LIN {X 0,Y 483.427,Z 781.933,A -85,B 0,C 180,E1 -6916.12,E2 -6916.12} C_VEL
LIN {X 0,Y 482.975,Z 793.62,A -85,B 0,C 180,E1 -6916.772,E2 -6916.772} C_VEL
LIN {X 0,Y 482.538,Z 805.095,A -85,B 0,C 180,E1 -6917.594,E2 -6917.594} C_VEL
LIN {X 0,Y 482.15,Z 815.757,A -85,B 0,C 180,E1 -6918.544,E2 -6918.544} C_VEL
LIN {X 0,Y 481.803,Z 824.454,A -85,B 0,C 180,E1 -6919.494,E2 -6919.494} C_VEL
LIN {X 0,Y 481.522,Z 832.495,A -85,B 0,C 180,E1 -6920.549,E2 -6920.549} C_VEL
LIN {X 0,Y 481.338,Z 839.236,A -85,B 0,C 180,E1 -6921.604,E2 -6921.604} C_VEL
LIN {X 0,Y 481.117,Z 845.911,A -85,B 0,C 180,E1 -6922.867,E2 -6922.867} C_VEL
LIN {X 0,Y 481.068,Z 851.207,A -85,B 0,C 180,E1 -6924.13,E2 -6924.13} C_VEL
LIN {X 0,Y 480.941,Z 855.277,A -85,B 0,C 180,E1 -6925.39,E2 -6925.39} C_VEL
LIN {X 0,Y 480.957,Z 858.306,A -85,B 0,C 180,E1 -6926.649,E2 -6926.649} C_VEL
LIN {X 0,Y 480.902,Z 859.812,A -85,B 0,C 180,E1 -6927.487,E2 -6927.487} C_VEL
LIN {X 0,Y 480.86,Z 861.418,A -85,B 0,C 180,E1 -6929.162,E2 -6929.162} C_VEL
LIN {X 0,Y 480.844,Z 861.684,A -85,B 0,C 180,E1 -6930,E2 -6930} C_VEL
LIN {X 0,Y 480.855,Z 861.455,A -85,B 0,C 180,E1 -6930.837,E2 -6930.837} C_VEL
LIN {X 0,Y 480.902,Z 859.817,A -85,B 0,C 180,E1 -6932.512,E2 -6932.512} C_VEL
LIN {X 0,Y 480.955,Z 858.409,A -85,B 0,C 180,E1 -6933.35,E2 -6933.35} C_VEL
LIN {X 0,Y 480.94,Z 855.356,A -85,B 0,C 180,E1 -6934.609,E2 -6934.609} C_VEL
LIN {X 0,Y 481.067,Z 851.27,A -85,B 0,C 180,E1 -6935.869,E2 -6935.869} C_VEL
LIN {X 0,Y 481.15,Z 845.081,A -85,B 0,C 180,E1 -6937.342,E2 -6937.342} C_VEL
LIN {X 0,Y 481.372,Z 838.203,A -85,B 0,C 180,E1 -6938.606,E2 -6938.606} C_VEL
LIN {X 0,Y 481.64,Z 829.782,A -85,B 0,C 180,E1 -6939.872,E2 -6939.872} C_VEL
LIN {X 0,Y 481.945,Z 821.073,A -85,B 0,C 180,E1 -6940.927,E2 -6940.927} C_VEL
LIN {X 0,Y 482.433,Z 810.454,A -85,B 0,C 180,E1 -6941.981,E2 -6941.981} C_VEL
LIN {X 0,Y 482.803,Z 798.946,A -85,B 0,C 180,E1 -6942.9,E2 -6942.9} C_VEL
LIN {X 0,Y 483.277,Z 786.489,A -85,B 0,C 180,E1 -6943.669,E2 -6943.669} C_VEL
LIN {X 0,Y 483.656,Z 774.047,A -85,B 0,C 180,E1 -6944.247,E2 -6944.247} C_VEL
LIN {X 0,Y 483.668,Z 767.501,A -85,B 0,C 180,E1 -6944.489,E2 -6944.489} C_VEL
LIN {X 0,Y 482.005,Z 754.779,A -85,B 0,C 180,E1 -6944.877,E2 -6944.877} C_VEL
LIN {X 0,Y 481.559,Z 749.951,A -85,B 0,C 180,E1 -6944.986,E2 -6944.986} C_VEL
LIN {X 0,Y 481.886,Z 734.845,A -85,B 0,C 180,E1 -6948.206,E2 -6948.206} C_VEL
LIN {X 0,Y 482.217,Z 720.246,A -85,B 0,C 180,E1 -6951.367,E2 -6951.367} C_VEL
LIN {X 0,Y 482.622,Z 704.896,A -85,B 0,C 180,E1 -6954.749,E2 -6954.749} C_VEL
LIN {X 0,Y 483.035,Z 691.607,A -85,B 0,C 180,E1 -6957.748,E2 -6957.748} C_VEL
LIN {X 0,Y 483.624,Z 676.701,A -85,B 0,C 180,E1 -6961.205,E2 -6961.205} C_VEL
LIN {X 0,Y 484.172,Z 663.094,A -85,B 0,C 180,E1 -6964.478,E2 -6964.478} C_VEL
LIN {X 0,Y 484.454,Z 654.94,A -85,B 0,C 180,E1 -6966.497,E2 -6966.497} C_VEL
LIN {X 0,Y 482.901,Z 646.667,A -85,B 0,C 180,E1 -6968.741,E2 -6968.741} C_VEL
LIN {X 0,Y 481.668,Z 640.49,A -85,B 0,C 180,E1 -6970.52,E2 -6970.52} C_VEL
LIN {X 0,Y 481.637,Z 640.491,A -85,B 0,C 180,E1 -6973.299,E2 -6973.299} C_VEL
LIN {X 0,Y 481.682,Z 640.488,A -85,B 0,C 180,E1 -6976.705,E2 -6976.705} C_VEL
LIN {X 0,Y 481.69,Z 640.485,A -85,B 0,C 180,E1 -6980.061,E2 -6980.061} C_VEL
LIN {X 0,Y 481.634,Z 640.491,A -85,B 0,C 180,E1 -6982.203,E2 -6982.203} C_VEL
LIN {X 0,Y 481.688,Z 640.479,A -85,B 0,C 180,E1 -6985.318,E2 -6985.318} C_VEL
LIN {X 0,Y 481.644,Z 640.487,A -85,B 0,C 180,E1 -6988.311,E2 -6988.311} C_VEL
LIN {X 0,Y 481.703,Z 640.479,A -85,B 0,C 180,E1 -6991.219,E2 -6991.219} C_VEL
LIN {X 0,Y 481.702,Z 640.479,A -85,B 0,C 180,E1 -6994.043,E2 -6994.043} C_VEL
LIN {X 0,Y 481.67,Z 640.483,A -85,B 0,C 180,E1 -6996.811,E2 -6996.811} C_VEL
LIN {X 0,Y 481.692,Z 640.483,A -85,B 0,C 180,E1 -6999.502,E2 -6999.502} C_VEL
LIN {X 0,Y 481.702,Z 640.478,A -85,B 0,C 180,E1 -7002.158,E2 -7002.158} C_VEL
LIN {X 0,Y 481.737,Z 640.479,A -85,B 0,C 180,E1 -7004.775,E2 -7004.775} C_VEL
LIN {X 0,Y 481.791,Z 640.47,A -85,B 0,C 180,E1 -7008.216,E2 -7008.216} C_VEL
LIN {X 0,Y 481.759,Z 640.473,A -85,B 0,C 180,E1 -7011.611,E2 -7011.611} C_VEL
LIN {X 0,Y 481.811,Z 640.47,A -85,B 0,C 180,E1 -7014.139,E2 -7014.139} C_VEL
LIN {X 0,Y 481.923,Z 640.453,A -85,B 0,C 180,E1 -7017.492,E2 -7017.492} C_VEL
LIN {X 0,Y 481.9,Z 640.459,A -85,B 0,C 180,E1 -7020.836,E2 -7020.836} C_VEL
LIN {X 0,Y 481.924,Z 640.458,A -85,B 0,C 180,E1 -7022.507,E2 -7022.507} C_VEL
LIN {X 0,Y 481.743,Z 640.595,A -85,B 0,C 180,E1 -7023.555,E2 -7023.555} C_VEL
LIN {X 0,Y 482.624,Z 646.304,A -85,B 0,C 180,E1 -7025.012,E2 -7025.012} C_VEL
LIN {X 0,Y 482.79,Z 656.329,A -85,B 0,C 180,E1 -7027.528,E2 -7027.528} C_VEL
LIN {X 0,Y 482.659,Z 667.926,A -85,B 0,C 180,E1 -7030.487,E2 -7030.487} C_VEL
LIN {X 0,Y 482.588,Z 677.613,A -85,B 0,C 180,E1 -7033.003,E2 -7033.003} C_VEL
LIN {X 0,Y 482.37,Z 689.295,A -85,B 0,C 180,E1 -7036.071,E2 -7036.071} C_VEL
LIN {X 0,Y 482.136,Z 700.788,A -85,B 0,C 180,E1 -7039.146,E2 -7039.146} C_VEL
LIN {X 0,Y 481.9,Z 712.481,A -85,B 0,C 180,E1 -7042.283,E2 -7042.283} C_VEL
LIN {X 0,Y 481.666,Z 724.354,A -85,B 0,C 180,E1 -7045.504,E2 -7045.504} C_VEL
LIN {X 0,Y 481.595,Z 726.474,A -85,B 0,C 180,E1 -7046.079,E2 -7046.079} C_VEL
LIN {X 0,Y 484.069,Z 741.262,A -85,B 0,C 180,E1 -7046.545,E2 -7046.545} C_VEL
LIN {X 0,Y 483.708,Z 754.433,A -85,B 0,C 180,E1 -7047.052,E2 -7047.052} C_VEL
LIN {X 0,Y 483.248,Z 767.048,A -85,B 0,C 180,E1 -7047.735,E2 -7047.735} C_VEL
LIN {X 0,Y 482.824,Z 779.115,A -85,B 0,C 180,E1 -7048.589,E2 -7048.589} C_VEL
LIN {X 0,Y 482.382,Z 789.501,A -85,B 0,C 180,E1 -7049.524,E2 -7049.524} C_VEL
LIN {X 0,Y 481.935,Z 799.526,A -85,B 0,C 180,E1 -7050.641,E2 -7050.641} C_VEL
LIN {X 0,Y 481.601,Z 807.216,A -85,B 0,C 180,E1 -7051.692,E2 -7051.692} C_VEL
LIN {X 0,Y 481.345,Z 814.641,A -85,B 0,C 180,E1 -7052.932,E2 -7052.932} C_VEL
LIN {X 0,Y 481.11,Z 820.823,A -85,B 0,C 180,E1 -7054.222,E2 -7054.222} C_VEL
LIN {X 0,Y 480.916,Z 826.562,A -85,B 0,C 180,E1 -7055.771,E2 -7055.771} C_VEL
LIN {X 0,Y 480.832,Z 829.462,A -85,B 0,C 180,E1 -7056.818,E2 -7056.818} C_VEL
LIN {X 0,Y 480.783,Z 831.725,A -85,B 0,C 180,E1 -7057.875,E2 -7057.875} C_VEL
LIN {X 0,Y 480.702,Z 833.614,A -85,B 0,C 180,E1 -7059.208,E2 -7059.208} C_VEL
LIN {X 0,Y 480.658,Z 834.484,A -85,B 0,C 180,E1 -7060.508,E2 -7060.508} C_VEL
LIN {X 0,Y 480.685,Z 834.413,A -85,B 0,C 180,E1 -7061.785,E2 -7061.785} C_VEL
LIN {X 0,Y 480.698,Z 832.973,A -85,B 0,C 180,E1 -7063.406,E2 -7063.406} C_VEL
LIN {X 0,Y 480.847,Z 830.113,A -85,B 0,C 180,E1 -7064.998,E2 -7064.998} C_VEL
LIN {X 0,Y 480.928,Z 826.941,A -85,B 0,C 180,E1 -7066.185,E2 -7066.185} C_VEL
LIN {X 0,Y 481.052,Z 822.862,A -85,B 0,C 180,E1 -7067.36,E2 -7067.36} C_VEL
LIN {X 0,Y 481.177,Z 817.743,A -85,B 0,C 180,E1 -7068.539,E2 -7068.539} C_VEL
LIN {X 0,Y 481.468,Z 810.441,A -85,B 0,C 180,E1 -7069.883,E2 -7069.883} C_VEL
LIN {X 0,Y 481.805,Z 801.756,A -85,B 0,C 180,E1 -7071.155,E2 -7071.155} C_VEL
LIN {X 0,Y 482.202,Z 792.467,A -85,B 0,C 180,E1 -7072.256,E2 -7072.256} C_VEL
LIN {X 0,Y 482.643,Z 782.457,A -85,B 0,C 180,E1 -7073.214,E2 -7073.214} C_VEL
LIN {X 0,Y 483.059,Z 771.967,A -85,B 0,C 180,E1 -7074.027,E2 -7074.027} C_VEL
LIN {X 0,Y 483.552,Z 759.705,A -85,B 0,C 180,E1 -7074.774,E2 -7074.774} C_VEL
LIN {X 0,Y 483.802,Z 750.922,A -85,B 0,C 180,E1 -7075.188,E2 -7075.188} C_VEL
LIN {X 0,Y 483.217,Z 747.306,A -85,B 0,C 180,E1 -7075.36,E2 -7075.36} C_VEL
LIN {X 0,Y 481.631,Z 743.95,A -85,B 0,C 180,E1 -7075.54,E2 -7075.54} C_VEL
LIN {X 0,Y 476.928,Z 736.321,A -85,B 0,C 180,E1 -7075.926,E2 -7075.926} C_VEL
LIN {X 0,Y 475.668,Z 732.622,A -85,B 0,C 180,E1 -7076.054,E2 -7076.054} C_VEL
LIN {X 0,Y 474.549,Z 726.5,A -85,B 0,C 180,E1 -7076.238,E2 -7076.238} C_VEL
LIN {X 0,Y 474.82,Z 714.749,A -85,B 0,C 180,E1 -7079.469,E2 -7079.469} C_VEL
LIN {X 0,Y 475.098,Z 704.87,A -85,B 0,C 180,E1 -7082.202,E2 -7082.202} C_VEL
LIN {X 0,Y 475.378,Z 694.436,A -85,B 0,C 180,E1 -7085.081,E2 -7085.081} C_VEL
LIN {X 0,Y 475.689,Z 682.671,A -85,B 0,C 180,E1 -7088.325,E2 -7088.325} C_VEL
LIN {X 0,Y 475.933,Z 671.182,A -85,B 0,C 180,E1 -7091.49,E2 -7091.49} C_VEL
LIN {X 0,Y 476.149,Z 659.898,A -85,B 0,C 180,E1 -7094.593,E2 -7094.593} C_VEL
LIN {X 0,Y 476.103,Z 650.411,A -85,B 0,C 180,E1 -7097.208,E2 -7097.208} C_VEL
LIN {X 0,Y 475.298,Z 644.411,A -85,B 0,C 180,E1 -7098.918,E2 -7098.918} C_VEL
LIN {X 0,Y 474.693,Z 641.359,A -85,B 0,C 180,E1 -7099.821,E2 -7099.821} C_VEL
LIN {X 0,Y 474.786,Z 641.347,A -85,B 0,C 180,E1 -7102.642,E2 -7102.642} C_VEL
LIN {X 0,Y 474.755,Z 641.351,A -85,B 0,C 180,E1 -7104.905,E2 -7104.905} C_VEL
LIN {X 0,Y 474.896,Z 641.333,A -85,B 0,C 180,E1 -7107.456,E2 -7107.456} C_VEL
LIN {X 0,Y 474.914,Z 641.329,A -85,B 0,C 180,E1 -7110,E2 -7110} C_VEL
LIN {X 0,Y 474.896,Z 641.331,A -85,B 0,C 180,E1 -7112.545,E2 -7112.545} C_VEL
LIN {X 0,Y 474.772,Z 641.348,A -85,B 0,C 180,E1 -7115.948,E2 -7115.948} C_VEL
LIN {X 0,Y 474.73,Z 641.353,A -85,B 0,C 180,E1 -7118.514,E2 -7118.514} C_VEL
LIN {X 0,Y 474.741,Z 641.349,A -85,B 0,C 180,E1 -7121.962,E2 -7121.962} C_VEL
LIN {X 0,Y 474.683,Z 641.358,A -85,B 0,C 180,E1 -7125.768,E2 -7125.768} C_VEL
LIN {X 0,Y 474.667,Z 641.361,A -85,B 0,C 180,E1 -7129.01,E2 -7129.01} C_VEL
LIN {X 0,Y 474.589,Z 641.371,A -85,B 0,C 180,E1 -7131.729,E2 -7131.729} C_VEL
LIN {X 0,Y 474.649,Z 641.364,A -85,B 0,C 180,E1 -7133.652,E2 -7133.652} C_VEL
LIN {X 0,Y 477.203,Z 650.814,A -85,B 0,C 180,E1 -7134.238,E2 -7134.238} C_VEL
LIN {X 0,Y 476.972,Z 661.909,A -85,B 0,C 180,E1 -7134.947,E2 -7134.947} C_VEL
LIN {X 0,Y 476.498,Z 673.39,A -85,B 0,C 180,E1 -7135.881,E2 -7135.881} C_VEL
LIN {X 0,Y 476.09,Z 683.215,A -85,B 0,C 180,E1 -7136.878,E2 -7136.878} C_VEL
LIN {X 0,Y 475.726,Z 692.476,A -85,B 0,C 180,E1 -7138.038,E2 -7138.038} C_VEL
LIN {X 0,Y 475.342,Z 700.4,A -85,B 0,C 180,E1 -7139.27,E2 -7139.27} C_VEL
LIN {X 0,Y 475.043,Z 706.99,A -85,B 0,C 180,E1 -7140.538,E2 -7140.538} C_VEL
LIN {X 0,Y 474.802,Z 711.876,A -85,B 0,C 180,E1 -7141.7,E2 -7141.7} C_VEL
LIN {X 0,Y 474.595,Z 716.839,A -85,B 0,C 180,E1 -7143.224,E2 -7143.224} C_VEL
LIN {X 0,Y 474.467,Z 719.337,A -85,B 0,C 180,E1 -7144.255,E2 -7144.255} C_VEL
LIN {X 0,Y 474.365,Z 721.447,A -85,B 0,C 180,E1 -7145.427,E2 -7145.427} C_VEL
LIN {X 0,Y 474.285,Z 722.963,A -85,B 0,C 180,E1 -7146.853,E2 -7146.853} C_VEL
LIN {X 0,Y 474.312,Z 723.349,A -85,B 0,C 180,E1 -7148.486,E2 -7148.486} C_VEL
LIN {X 0,Y 474.353,Z 722.79,A -85,B 0,C 180,E1 -7149.607,E2 -7149.607} C_VEL
LIN {X 0,Y 474.425,Z 721.256,A -85,B 0,C 180,E1 -7150.931,E2 -7150.931} C_VEL
LIN {X 0,Y 474.576,Z 718.785,A -85,B 0,C 180,E1 -7152.23,E2 -7152.23} C_VEL
LIN {X 0,Y 474.751,Z 715.391,A -85,B 0,C 180,E1 -7153.5,E2 -7153.5} C_VEL
LIN {X 0,Y 474.957,Z 710.197,A -85,B 0,C 180,E1 -7154.952,E2 -7154.952} C_VEL
LIN {X 0,Y 475.317,Z 703.304,A -85,B 0,C 180,E1 -7156.428,E2 -7156.428} C_VEL
LIN {X 0,Y 475.677,Z 696.215,A -85,B 0,C 180,E1 -7157.624,E2 -7157.624} C_VEL
LIN {X 0,Y 476.057,Z 687.294,A -85,B 0,C 180,E1 -7158.843,E2 -7158.843} C_VEL
LIN {X 0,Y 476.534,Z 678.215,A -85,B 0,C 180,E1 -7159.848,E2 -7159.848} C_VEL
LIN {X 0,Y 476.893,Z 668.033,A -85,B 0,C 180,E1 -7160.769,E2 -7160.769} C_VEL
LIN {X 0,Y 477.24,Z 656.015,A -85,B 0,C 180,E1 -7161.62,E2 -7161.62} C_VEL
LIN {X 0,Y 477.318,Z 650.683,A -85,B 0,C 180,E1 -7161.934,E2 -7161.934} C_VEL
LIN {X 0,Y 474.626,Z 641.364,A -85,B 0,C 180,E1 -7162.519,E2 -7162.519} C_VEL
LIN {X 0,Y 474.638,Z 641.362,A -85,B 0,C 180,E1 -7166.016,E2 -7166.016} C_VEL
LIN {X 0,Y 474.605,Z 641.367,A -85,B 0,C 180,E1 -7169.19,E2 -7169.19} C_VEL
LIN {X 0,Y 474.647,Z 641.365,A -85,B 0,C 180,E1 -7171.718,E2 -7171.718} C_VEL
LIN {X 0,Y 474.652,Z 641.356,A -85,B 0,C 180,E1 -7174.583,E2 -7174.583} C_VEL
LIN {X 0,Y 474.601,Z 641.362,A -85,B 0,C 180,E1 -7177.355,E2 -7177.355} C_VEL
LIN {X 0,Y 474.656,Z 641.361,A -85,B 0,C 180,E1 -7180.09,E2 -7180.09} C_VEL
LIN {X 0,Y 474.651,Z 641.356,A -85,B 0,C 180,E1 -7182.775,E2 -7182.775} C_VEL
LIN {X 0,Y 474.649,Z 641.36,A -85,B 0,C 180,E1 -7185.421,E2 -7185.421} C_VEL
LIN {X 0,Y 474.705,Z 641.354,A -85,B 0,C 180,E1 -7188.038,E2 -7188.038} C_VEL
LIN {X 0,Y 474.729,Z 641.349,A -85,B 0,C 180,E1 -7191.487,E2 -7191.487} C_VEL
LIN {X 0,Y 474.78,Z 641.347,A -85,B 0,C 180,E1 -7194.053,E2 -7194.053} C_VEL
LIN {X 0,Y 474.896,Z 641.323,A -85,B 0,C 180,E1 -7197.456,E2 -7197.456} C_VEL
LIN {X 0,Y 474.913,Z 641.328,A -85,B 0,C 180,E1 -7200,E2 -7200} C_VEL
LIN {X 0,Y 474.896,Z 641.328,A -85,B 0,C 180,E1 -7202.545,E2 -7202.545} C_VEL
LIN {X 0,Y 474.78,Z 641.341,A -85,B 0,C 180,E1 -7205.948,E2 -7205.948} C_VEL
LIN {X 0,Y 474.73,Z 641.346,A -85,B 0,C 180,E1 -7208.514,E2 -7208.514} C_VEL
LIN {X 0,Y 474.706,Z 641.354,A -85,B 0,C 180,E1 -7211.963,E2 -7211.963} C_VEL
LIN {X 0,Y 474.701,Z 641.35,A -85,B 0,C 180,E1 -7215.456,E2 -7215.456} C_VEL
LIN {X 0,Y 474.666,Z 641.354,A -85,B 0,C 180,E1 -7219.01,E2 -7219.01} C_VEL
LIN {X 0,Y 474.59,Z 641.365,A -85,B 0,C 180,E1 -7221.729,E2 -7221.729} C_VEL
LIN {X 0,Y 474.659,Z 641.362,A -85,B 0,C 180,E1 -7224.493,E2 -7224.493} C_VEL
LIN {X 0,Y 474.683,Z 641.353,A -85,B 0,C 180,E1 -7227.334,E2 -7227.334} C_VEL
LIN {X 0,Y 474.607,Z 641.367,A -85,B 0,C 180,E1 -7230.23,E2 -7230.23} C_VEL
LIN {X 0,Y 474.645,Z 641.36,A -85,B 0,C 180,E1 -7233.22,E2 -7233.22} C_VEL
LIN {X 0,Y 474.591,Z 641.371,A -85,B 0,C 180,E1 -7236.324,E2 -7236.324} C_VEL
LIN {X 0,Y 474.63,Z 641.361,A -85,B 0,C 180,E1 -7239.648,E2 -7239.648} C_VEL
LIN {X 0,Y 474.618,Z 641.363,A -85,B 0,C 180,E1 -7242.934,E2 -7242.934} C_VEL
LIN {X 0,Y 474.612,Z 641.365,A -85,B 0,C 180,E1 -7245.895,E2 -7245.895} C_VEL
LIN {X 0,Y 474.63,Z 641.372,A -85,B 0,C 180,E1 -7249.041,E2 -7249.041} C_VEL
LIN {X 0,Y 474.648,Z 641.378,A -85,B 0,C 180,E1 -7249.799,E2 -7249.799} C_VEL
LIN {X 0,Y 476.716,Z 652.009,A -85,B 0,C 180,E1 -7252.811,E2 -7252.811} C_VEL
LIN {X 0,Y 477.086,Z 656.071,A -85,B 0,C 180,E1 -7253.896,E2 -7253.896} C_VEL
LIN {X 0,Y 476.52,Z 669.453,A -85,B 0,C 180,E1 -7257.211,E2 -7257.211} C_VEL
LIN {X 0,Y 476.074,Z 682.373,A -85,B 0,C 180,E1 -7260.276,E2 -7260.276} C_VEL
LIN {X 0,Y 475.643,Z 697.254,A -85,B 0,C 180,E1 -7263.687,E2 -7263.687} C_VEL
LIN {X 0,Y 475.306,Z 709.747,A -85,B 0,C 180,E1 -7266.47,E2 -7266.47} C_VEL
LIN {X 0,Y 474.934,Z 725.361,A -85,B 0,C 180,E1 -7269.876,E2 -7269.876} C_VEL
LIN {X 0,Y 474.656,Z 738.834,A -85,B 0,C 180,E1 -7272.774,E2 -7272.774} C_VEL
LIN {X 0,Y 474.456,Z 748.246,A -85,B 0,C 180,E1 -7274.783,E2 -7274.783} C_VEL
LIN {X 0,Y 475.885,Z 762.604,A -85,B 0,C 180,E1 -7275.172,E2 -7275.172} C_VEL
LIN {X 0,Y 476.883,Z 769.641,A -85,B 0,C 180,E1 -7275.436,E2 -7275.436} C_VEL
LIN {X 0,Y 476.45,Z 781.864,A -85,B 0,C 180,E1 -7275.968,E2 -7275.968} C_VEL
LIN {X 0,Y 475.937,Z 794.279,A -85,B 0,C 180,E1 -7276.692,E2 -7276.692} C_VEL
LIN {X 0,Y 475.441,Z 808.391,A -85,B 0,C 180,E1 -7277.757,E2 -7277.757} C_VEL
LIN {X 0,Y 475.06,Z 818.329,A -85,B 0,C 180,E1 -7278.695,E2 -7278.695} C_VEL
LIN {X 0,Y 474.646,Z 827.581,A -85,B 0,C 180,E1 -7279.765,E2 -7279.765} C_VEL
LIN {X 0,Y 474.326,Z 836.509,A -85,B 0,C 180,E1 -7281.049,E2 -7281.049} C_VEL
LIN {X 0,Y 474.11,Z 843.623,A -85,B 0,C 180,E1 -7282.333,E2 -7282.333} C_VEL
LIN {X 0,Y 473.982,Z 849.619,A -85,B 0,C 180,E1 -7283.687,E2 -7283.687} C_VEL
LIN {X 0,Y 473.908,Z 853.793,A -85,B 0,C 180,E1 -7284.895,E2 -7284.895} C_VEL
LIN {X 0,Y 473.883,Z 858.008,A -85,B 0,C 180,E1 -7286.599,E2 -7286.599} C_VEL
LIN {X 0,Y 473.816,Z 859.477,A -85,B 0,C 180,E1 -7287.449,E2 -7287.449} C_VEL
LIN {X 0,Y 473.783,Z 861.076,A -85,B 0,C 180,E1 -7289.15,E2 -7289.15} C_VEL
LIN {X 0,Y 473.765,Z 861.311,A -85,B 0,C 180,E1 -7290,E2 -7290} C_VEL
LIN {X 0,Y 473.778,Z 861.086,A -85,B 0,C 180,E1 -7290.849,E2 -7290.849} C_VEL
LIN {X 0,Y 473.815,Z 859.441,A -85,B 0,C 180,E1 -7292.55,E2 -7292.55} C_VEL
LIN {X 0,Y 473.88,Z 858.008,A -85,B 0,C 180,E1 -7293.4,E2 -7293.4} C_VEL
LIN {X 0,Y 473.855,Z 854.979,A -85,B 0,C 180,E1 -7294.679,E2 -7294.679} C_VEL
LIN {X 0,Y 473.967,Z 850.886,A -85,B 0,C 180,E1 -7295.957,E2 -7295.957} C_VEL
LIN {X 0,Y 474.041,Z 845.631,A -85,B 0,C 180,E1 -7297.239,E2 -7297.239} C_VEL
LIN {X 0,Y 474.31,Z 837.736,A -85,B 0,C 180,E1 -7298.735,E2 -7298.735} C_VEL
LIN {X 0,Y 474.577,Z 829.128,A -85,B 0,C 180,E1 -7300.02,E2 -7300.02} C_VEL
LIN {X 0,Y 474.944,Z 820.219,A -85,B 0,C 180,E1 -7301.09,E2 -7301.09} C_VEL
LIN {X 0,Y 475.467,Z 808.63,A -85,B 0,C 180,E1 -7302.232,E2 -7302.232} C_VEL
LIN {X 0,Y 475.842,Z 797.489,A -85,B 0,C 180,E1 -7303.125,E2 -7303.125} C_VEL
LIN {X 0,Y 476.323,Z 785.478,A -85,B 0,C 180,E1 -7303.872,E2 -7303.872} C_VEL
LIN {X 0,Y 476.758,Z 773.046,A -85,B 0,C 180,E1 -7304.458,E2 -7304.458} C_VEL
LIN {X 0,Y 476.678,Z 768.01,A -85,B 0,C 180,E1 -7304.651,E2 -7304.651} C_VEL
LIN {X 0,Y 475.117,Z 755.564,A -85,B 0,C 180,E1 -7305.057,E2 -7305.057} C_VEL
LIN {X 0,Y 474.48,Z 748.962,A -85,B 0,C 180,E1 -7305.215,E2 -7305.215} C_VEL
LIN {X 0,Y 474.834,Z 734.329,A -85,B 0,C 180,E1 -7308.399,E2 -7308.399} C_VEL
LIN {X 0,Y 475.18,Z 719.4,A -85,B 0,C 180,E1 -7311.7,E2 -7311.7} C_VEL
LIN {X 0,Y 475.642,Z 704.092,A -85,B 0,C 180,E1 -7315.138,E2 -7315.138} C_VEL
LIN {X 0,Y 476.154,Z 689.845,A -85,B 0,C 180,E1 -7318.424,E2 -7318.424} C_VEL
LIN {X 0,Y 476.668,Z 676.506,A -85,B 0,C 180,E1 -7321.586,E2 -7321.586} C_VEL
LIN {X 0,Y 477.261,Z 663.804,A -85,B 0,C 180,E1 -7324.692,E2 -7324.692} C_VEL
LIN {X 0,Y 477.51,Z 656.299,A -85,B 0,C 180,E1 -7326.589,E2 -7326.589} C_VEL
LIN {X 0,Y 475.93,Z 647.787,A -85,B 0,C 180,E1 -7328.932,E2 -7328.932} C_VEL
LIN {X 0,Y 474.624,Z 641.367,A -85,B 0,C 180,E1 -7330.807,E2 -7330.807} C_VEL
LIN {X 0,Y 474.607,Z 641.367,A -85,B 0,C 180,E1 -7334.104,E2 -7334.104} C_VEL
LIN {X 0,Y 474.65,Z 641.361,A -85,B 0,C 180,E1 -7337.069,E2 -7337.069} C_VEL
LIN {X 0,Y 474.671,Z 641.361,A -85,B 0,C 180,E1 -7340.457,E2 -7340.457} C_VEL
LIN {X 0,Y 474.589,Z 641.366,A -85,B 0,C 180,E1 -7343.676,E2 -7343.676} C_VEL
LIN {X 0,Y 474.639,Z 641.36,A -85,B 0,C 180,E1 -7346.779,E2 -7346.779} C_VEL
LIN {X 0,Y 474.61,Z 641.368,A -85,B 0,C 180,E1 -7349.77,E2 -7349.77} C_VEL
LIN {X 0,Y 474.71,Z 641.351,A -85,B 0,C 180,E1 -7352.68,E2 -7352.68} C_VEL
LIN {X 0,Y 474.655,Z 641.362,A -85,B 0,C 180,E1 -7355.507,E2 -7355.507} C_VEL
LIN {X 0,Y 474.666,Z 641.361,A -85,B 0,C 180,E1 -7359.185,E2 -7359.185} C_VEL
LIN {X 0,Y 474.652,Z 641.357,A -85,B 0,C 180,E1 -7361.884,E2 -7361.884} C_VEL
LIN {X 0,Y 474.694,Z 641.354,A -85,B 0,C 180,E1 -7364.544,E2 -7364.544} C_VEL
LIN {X 0,Y 474.734,Z 641.348,A -85,B 0,C 180,E1 -7368.038,E2 -7368.038} C_VEL
LIN {X 0,Y 474.724,Z 641.35,A -85,B 0,C 180,E1 -7371.486,E2 -7371.486} C_VEL
LIN {X 0,Y 474.773,Z 641.346,A -85,B 0,C 180,E1 -7374.052,E2 -7374.052} C_VEL
LIN {X 0,Y 474.889,Z 641.33,A -85,B 0,C 180,E1 -7377.455,E2 -7377.455} C_VEL
LIN {X 0,Y 474.906,Z 641.333,A -85,B 0,C 180,E1 -7380,E2 -7380} C_VEL
LIN {X 0,Y 474.793,Z 641.346,A -85,B 0,C 180,E1 -7382.97,E2 -7382.97} C_VEL
LIN {X 0,Y 474.714,Z 641.474,A -85,B 0,C 180,E1 -7383.342,E2 -7383.342} C_VEL
LIN {X 0,Y 475.713,Z 648.213,A -85,B 0,C 180,E1 -7385.085,E2 -7385.085} C_VEL
LIN {X 0,Y 475.877,Z 659.654,A -85,B 0,C 180,E1 -7387.995,E2 -7387.995} C_VEL
LIN {X 0,Y 475.683,Z 671.596,A -85,B 0,C 180,E1 -7391.073,E2 -7391.073} C_VEL
LIN {X 0,Y 475.558,Z 681.428,A -85,B 0,C 180,E1 -7393.677,E2 -7393.677} C_VEL
LIN {X 0,Y 475.281,Z 693.027,A -85,B 0,C 180,E1 -7396.759,E2 -7396.759} C_VEL
LIN {X 0,Y 475.088,Z 703.087,A -85,B 0,C 180,E1 -7399.441,E2 -7399.441} C_VEL
LIN {X 0,Y 474.873,Z 713.146,A -85,B 0,C 180,E1 -7402.172,E2 -7402.172} C_VEL
LIN {X 0,Y 474.635,Z 725.093,A -85,B 0,C 180,E1 -7405.43,E2 -7405.43} C_VEL
LIN {X 0,Y 474.578,Z 726.717,A -85,B 0,C 180,E1 -7405.874,E2 -7405.874} C_VEL
LIN {X 0,Y 476.858,Z 739.805,A -85,B 0,C 180,E1 -7406.27,E2 -7406.27} C_VEL
LIN {X 0,Y 477.101,Z 745.206,A -85,B 0,C 180,E1 -7406.462,E2 -7406.462} C_VEL
LIN {X 0,Y 476.719,Z 757.96,A -85,B 0,C 180,E1 -7407.017,E2 -7407.017} C_VEL
LIN {X 0,Y 476.252,Z 769.703,A -85,B 0,C 180,E1 -7407.7,E2 -7407.7} C_VEL
LIN {X 0,Y 475.771,Z 781.216,A -85,B 0,C 180,E1 -7408.57,E2 -7408.57} C_VEL
LIN {X 0,Y 475.285,Z 791.752,A -85,B 0,C 180,E1 -7409.568,E2 -7409.568} C_VEL
LIN {X 0,Y 474.902,Z 800.886,A -85,B 0,C 180,E1 -7410.637,E2 -7410.637} C_VEL
LIN {X 0,Y 474.544,Z 808.47,A -85,B 0,C 180,E1 -7411.719,E2 -7411.719} C_VEL
LIN {X 0,Y 474.245,Z 815.881,A -85,B 0,C 180,E1 -7413.018,E2 -7413.018} C_VEL
LIN {X 0,Y 474.027,Z 821.72,A -85,B 0,C 180,E1 -7414.291,E2 -7414.291} C_VEL
LIN {X 0,Y 473.837,Z 827.27,A -85,B 0,C 180,E1 -7415.864,E2 -7415.864} C_VEL
LIN {X 0,Y 473.723,Z 831.226,A -85,B 0,C 180,E1 -7417.464,E2 -7417.464} C_VEL
LIN {X 0,Y 473.646,Z 833.056,A -85,B 0,C 180,E1 -7418.55,E2 -7418.55} C_VEL
LIN {X 0,Y 473.583,Z 834.247,A -85,B 0,C 180,E1 -7419.652,E2 -7419.652} C_VEL
LIN {X 0,Y 473.553,Z 834.739,A -85,B 0,C 180,E1 -7420.81,E2 -7420.81} C_VEL
LIN {X 0,Y 473.589,Z 834.442,A -85,B 0,C 180,E1 -7422.1,E2 -7422.1} C_VEL
LIN {X 0,Y 473.6,Z 833.28,A -85,B 0,C 180,E1 -7423.354,E2 -7423.354} C_VEL
LIN {X 0,Y 473.708,Z 831.27,A -85,B 0,C 180,E1 -7424.592,E2 -7424.592} C_VEL
LIN {X 0,Y 473.852,Z 827.189,A -85,B 0,C 180,E1 -7426.24,E2 -7426.24} C_VEL
LIN {X 0,Y 473.993,Z 823.051,A -85,B 0,C 180,E1 -7427.452,E2 -7427.452} C_VEL
LIN {X 0,Y 474.187,Z 816.667,A -85,B 0,C 180,E1 -7428.908,E2 -7428.908} C_VEL
LIN {X 0,Y 474.499,Z 809.738,A -85,B 0,C 180,E1 -7430.155,E2 -7430.155} C_VEL
LIN {X 0,Y 474.881,Z 800.946,A -85,B 0,C 180,E1 -7431.434,E2 -7431.434} C_VEL
LIN {X 0,Y 475.301,Z 791.388,A -85,B 0,C 180,E1 -7432.549,E2 -7432.549} C_VEL
LIN {X 0,Y 475.77,Z 781.131,A -85,B 0,C 180,E1 -7433.519,E2 -7433.519} C_VEL
LIN {X 0,Y 476.2,Z 770.288,A -85,B 0,C 180,E1 -7434.346,E2 -7434.346} C_VEL
LIN {X 0,Y 476.697,Z 758.702,A -85,B 0,C 180,E1 -7435.032,E2 -7435.032} C_VEL
LIN {X 0,Y 477.064,Z 746.239,A -85,B 0,C 180,E1 -7435.586,E2 -7435.586} C_VEL
LIN {X 0,Y 476.888,Z 740.191,A -85,B 0,C 180,E1 -7435.804,E2 -7435.804} C_VEL
LIN {X 0,Y 475.668,Z 732.622,A -85,B 0,C 180,E1 -7436.054,E2 -7436.054} C_VEL
LIN {X 0,Y 474.755,Z 729.411,A -85,B 0,C 180,E1 -7436.232,E2 -7436.232} C_VEL
LIN {X 0,Y 473.539,Z 726.86,A -85,B 0,C 180,E1 -7436.522,E2 -7436.522} C_VEL
LIN {X 0,Y 471.551,Z 723.981,A -85,B 0,C 180,E1 -7437.079,E2 -7437.079} C_VEL
LIN {X 0,Y 468.657,Z 720.158,A -85,B 0,C 180,E1 -7438.223,E2 -7438.223} C_VEL
LIN {X 0,Y 467.809,Z 717.693,A -85,B 0,C 180,E1 -7438.95,E2 -7438.95} C_VEL
LIN {X 0,Y 467.765,Z 716.828,A -85,B 0,C 180,E1 -7439.193,E2 -7439.193} C_VEL
LIN {X 0,Y 468.051,Z 707.57,A -85,B 0,C 180,E1 -7441.772,E2 -7441.772} C_VEL
LIN {X 0,Y 468.387,Z 695.378,A -85,B 0,C 180,E1 -7445.158,E2 -7445.158} C_VEL
LIN {X 0,Y 468.692,Z 683.766,A -85,B 0,C 180,E1 -7448.386,E2 -7448.386} C_VEL
LIN {X 0,Y 468.956,Z 673.558,A -85,B 0,C 180,E1 -7451.218,E2 -7451.218} C_VEL
LIN {X 0,Y 469.153,Z 662.248,A -85,B 0,C 180,E1 -7454.358,E2 -7454.358} C_VEL
LIN {X 0,Y 469.229,Z 652.675,A -85,B 0,C 180,E1 -7457.017,E2 -7457.017} C_VEL
LIN {X 0,Y 468.509,Z 646.6,A -85,B 0,C 180,E1 -7458.755,E2 -7458.755} C_VEL
LIN {X 0,Y 467.645,Z 642.236,A -85,B 0,C 180,E1 -7460.048,E2 -7460.048} C_VEL
LIN {X 0,Y 467.707,Z 642.229,A -85,B 0,C 180,E1 -7463.096,E2 -7463.096} C_VEL
LIN {X 0,Y 467.727,Z 642.226,A -85,B 0,C 180,E1 -7464.828,E2 -7464.828} C_VEL
LIN {X 0,Y 467.862,Z 642.209,A -85,B 0,C 180,E1 -7467.418,E2 -7467.418} C_VEL
LIN {X 0,Y 467.885,Z 642.205,A -85,B 0,C 180,E1 -7470,E2 -7470} C_VEL
LIN {X 0,Y 467.862,Z 642.207,A -85,B 0,C 180,E1 -7472.583,E2 -7472.583} C_VEL
LIN {X 0,Y 467.736,Z 642.223,A -85,B 0,C 180,E1 -7476.038,E2 -7476.038} C_VEL
LIN {X 0,Y 467.684,Z 642.232,A -85,B 0,C 180,E1 -7478.643,E2 -7478.643} C_VEL
LIN {X 0,Y 467.685,Z 642.229,A -85,B 0,C 180,E1 -7482.145,E2 -7482.145} C_VEL
LIN {X 0,Y 467.652,Z 642.233,A -85,B 0,C 180,E1 -7485.886,E2 -7485.886} C_VEL
LIN {X 0,Y 467.625,Z 642.24,A -85,B 0,C 180,E1 -7489.308,E2 -7489.308} C_VEL
LIN {X 0,Y 467.535,Z 642.251,A -85,B 0,C 180,E1 -7492.074,E2 -7492.074} C_VEL
LIN {X 0,Y 467.602,Z 642.242,A -85,B 0,C 180,E1 -7493.437,E2 -7493.437} C_VEL
LIN {X 0,Y 470.264,Z 651.794,A -85,B 0,C 180,E1 -7494.037,E2 -7494.037} C_VEL
LIN {X 0,Y 470.143,Z 662.657,A -85,B 0,C 180,E1 -7494.744,E2 -7494.744} C_VEL
LIN {X 0,Y 469.683,Z 673.211,A -85,B 0,C 180,E1 -7495.599,E2 -7495.599} C_VEL
LIN {X 0,Y 469.19,Z 684.072,A -85,B 0,C 180,E1 -7496.704,E2 -7496.704} C_VEL
LIN {X 0,Y 468.788,Z 693.855,A -85,B 0,C 180,E1 -7497.952,E2 -7497.952} C_VEL
LIN {X 0,Y 468.354,Z 702.206,A -85,B 0,C 180,E1 -7499.29,E2 -7499.29} C_VEL
LIN {X 0,Y 468.032,Z 709.221,A -85,B 0,C 180,E1 -7500.7,E2 -7500.7} C_VEL
LIN {X 0,Y 467.735,Z 714.979,A -85,B 0,C 180,E1 -7502.209,E2 -7502.209} C_VEL
LIN {X 0,Y 467.529,Z 719.446,A -85,B 0,C 180,E1 -7503.793,E2 -7503.793} C_VEL
LIN {X 0,Y 467.388,Z 721.586,A -85,B 0,C 180,E1 -7504.848,E2 -7504.848} C_VEL
LIN {X 0,Y 467.311,Z 723.146,A -85,B 0,C 180,E1 -7505.911,E2 -7505.911} C_VEL
LIN {X 0,Y 467.272,Z 724.158,A -85,B 0,C 180,E1 -7507.142,E2 -7507.142} C_VEL
LIN {X 0,Y 467.298,Z 724.363,A -85,B 0,C 180,E1 -7508.55,E2 -7508.55} C_VEL
LIN {X 0,Y 467.368,Z 723.194,A -85,B 0,C 180,E1 -7510.287,E2 -7510.287} C_VEL
LIN {X 0,Y 467.52,Z 720.49,A -85,B 0,C 180,E1 -7511.986,E2 -7511.986} C_VEL
LIN {X 0,Y 467.776,Z 716.007,A -85,B 0,C 180,E1 -7513.719,E2 -7513.719} C_VEL
LIN {X 0,Y 468.015,Z 711.04,A -85,B 0,C 180,E1 -7515.107,E2 -7515.107} C_VEL
LIN {X 0,Y 468.373,Z 704.555,A -85,B 0,C 180,E1 -7516.517,E2 -7516.517} C_VEL
LIN {X 0,Y 468.786,Z 696.869,A -85,B 0,C 180,E1 -7517.83,E2 -7517.83} C_VEL
LIN {X 0,Y 469.196,Z 688.126,A -85,B 0,C 180,E1 -7519.034,E2 -7519.034} C_VEL
LIN {X 0,Y 469.723,Z 678.584,A -85,B 0,C 180,E1 -7520.097,E2 -7520.097} C_VEL
LIN {X 0,Y 470.077,Z 668.249,A -85,B 0,C 180,E1 -7521.027,E2 -7521.027} C_VEL
LIN {X 0,Y 470.476,Z 655.968,A -85,B 0,C 180,E1 -7521.893,E2 -7521.893} C_VEL
LIN {X 0,Y 470.541,Z 652.416,A -85,B 0,C 180,E1 -7522.103,E2 -7522.103} C_VEL
LIN {X 0,Y 467.586,Z 642.241,A -85,B 0,C 180,E1 -7522.752,E2 -7522.752} C_VEL
LIN {X 0,Y 467.587,Z 642.24,A -85,B 0,C 180,E1 -7526.212,E2 -7526.212} C_VEL
LIN {X 0,Y 467.57,Z 642.244,A -85,B 0,C 180,E1 -7529.266,E2 -7529.266} C_VEL
LIN {X 0,Y 467.634,Z 642.232,A -85,B 0,C 180,E1 -7532.462,E2 -7532.462} C_VEL
LIN {X 0,Y 467.585,Z 642.238,A -85,B 0,C 180,E1 -7535.112,E2 -7535.112} C_VEL
LIN {X 0,Y 467.535,Z 642.247,A -85,B 0,C 180,E1 -7537.926,E2 -7537.926} C_VEL
LIN {X 0,Y 467.624,Z 642.233,A -85,B 0,C 180,E1 -7540.692,E2 -7540.692} C_VEL
LIN {X 0,Y 467.668,Z 642.232,A -85,B 0,C 180,E1 -7544.107,E2 -7544.107} C_VEL
LIN {X 0,Y 467.657,Z 642.234,A -85,B 0,C 180,E1 -7547.855,E2 -7547.855} C_VEL
LIN {X 0,Y 467.683,Z 642.226,A -85,B 0,C 180,E1 -7551.357,E2 -7551.357} C_VEL
LIN {X 0,Y 467.744,Z 642.222,A -85,B 0,C 180,E1 -7553.963,E2 -7553.963} C_VEL
LIN {X 0,Y 467.862,Z 642.199,A -85,B 0,C 180,E1 -7557.417,E2 -7557.417} C_VEL
LIN {X 0,Y 467.884,Z 642.203,A -85,B 0,C 180,E1 -7560,E2 -7560} C_VEL
LIN {X 0,Y 467.862,Z 642.204,A -85,B 0,C 180,E1 -7562.583,E2 -7562.583} C_VEL
LIN {X 0,Y 467.745,Z 642.219,A -85,B 0,C 180,E1 -7566.038,E2 -7566.038} C_VEL
LIN {X 0,Y 467.683,Z 642.223,A -85,B 0,C 180,E1 -7568.643,E2 -7568.643} C_VEL
LIN {X 0,Y 467.658,Z 642.233,A -85,B 0,C 180,E1 -7572.146,E2 -7572.146} C_VEL
LIN {X 0,Y 467.641,Z 642.231,A -85,B 0,C 180,E1 -7575.695,E2 -7575.695} C_VEL
LIN {X 0,Y 467.619,Z 642.234,A -85,B 0,C 180,E1 -7578.765,E2 -7578.765} C_VEL
LIN {X 0,Y 467.582,Z 642.237,A -85,B 0,C 180,E1 -7581.268,E2 -7581.268} C_VEL
LIN {X 0,Y 467.574,Z 642.239,A -85,B 0,C 180,E1 -7583.943,E2 -7583.943} C_VEL
LIN {X 0,Y 467.619,Z 642.237,A -85,B 0,C 180,E1 -7586.8,E2 -7586.8} C_VEL
LIN {X 0,Y 467.556,Z 642.241,A -85,B 0,C 180,E1 -7589.738,E2 -7589.738} C_VEL
LIN {X 0,Y 467.585,Z 642.243,A -85,B 0,C 180,E1 -7592.758,E2 -7592.758} C_VEL
LIN {X 0,Y 467.555,Z 642.244,A -85,B 0,C 180,E1 -7595.89,E2 -7595.89} C_VEL
LIN {X 0,Y 467.585,Z 642.241,A -85,B 0,C 180,E1 -7599.145,E2 -7599.145} C_VEL
LIN {X 0,Y 467.589,Z 642.241,A -85,B 0,C 180,E1 -7602.567,E2 -7602.567} C_VEL
LIN {X 0,Y 467.573,Z 642.246,A -85,B 0,C 180,E1 -7605.053,E2 -7605.053} C_VEL
LIN {X 0,Y 467.591,Z 642.244,A -85,B 0,C 180,E1 -7607.44,E2 -7607.44} C_VEL
LIN {X 0,Y 467.602,Z 642.328,A -85,B 0,C 180,E1 -7609.526,E2 -7609.526} C_VEL
LIN {X 0,Y 469.602,Z 652.502,A -85,B 0,C 180,E1 -7612.485,E2 -7612.485} C_VEL
LIN {X 0,Y 470.17,Z 657.423,A -85,B 0,C 180,E1 -7613.822,E2 -7613.822} C_VEL
LIN {X 0,Y 469.598,Z 669.786,A -85,B 0,C 180,E1 -7616.94,E2 -7616.94} C_VEL
LIN {X 0,Y 469.103,Z 681.881,A -85,B 0,C 180,E1 -7619.875,E2 -7619.875} C_VEL
LIN {X 0,Y 468.67,Z 695.274,A -85,B 0,C 180,E1 -7623.024,E2 -7623.024} C_VEL
LIN {X 0,Y 468.285,Z 708.779,A -85,B 0,C 180,E1 -7626.095,E2 -7626.095} C_VEL
LIN {X 0,Y 467.871,Z 724.33,A -85,B 0,C 180,E1 -7629.559,E2 -7629.559} C_VEL
LIN {X 0,Y 467.62,Z 737.739,A -85,B 0,C 180,E1 -7632.507,E2 -7632.507} C_VEL
LIN {X 0,Y 467.418,Z 747.12,A -85,B 0,C 180,E1 -7634.549,E2 -7634.549} C_VEL
LIN {X 0,Y 468.816,Z 762.347,A -85,B 0,C 180,E1 -7634.971,E2 -7634.971} C_VEL
LIN {X 0,Y 469.843,Z 771.236,A -85,B 0,C 180,E1 -7635.324,E2 -7635.324} C_VEL
LIN {X 0,Y 469.405,Z 783.794,A -85,B 0,C 180,E1 -7635.918,E2 -7635.918} C_VEL
LIN {X 0,Y 468.793,Z 798.021,A -85,B 0,C 180,E1 -7636.784,E2 -7636.784} C_VEL
LIN {X 0,Y 468.432,Z 809.671,A -85,B 0,C 180,E1 -7637.702,E2 -7637.702} C_VEL
LIN {X 0,Y 467.955,Z 820.109,A -85,B 0,C 180,E1 -7638.741,E2 -7638.741} C_VEL
LIN {X 0,Y 467.571,Z 828.989,A -85,B 0,C 180,E1 -7639.827,E2 -7639.827} C_VEL
LIN {X 0,Y 467.27,Z 836.298,A -85,B 0,C 180,E1 -7640.913,E2 -7640.913} C_VEL
LIN {X 0,Y 467.05,Z 843.459,A -85,B 0,C 180,E1 -7642.216,E2 -7642.216} C_VEL
LIN {X 0,Y 466.914,Z 848.816,A -85,B 0,C 180,E1 -7643.433,E2 -7643.433} C_VEL
LIN {X 0,Y 466.842,Z 853.587,A -85,B 0,C 180,E1 -7644.817,E2 -7644.817} C_VEL
LIN {X 0,Y 466.793,Z 857.83,A -85,B 0,C 180,E1 -7646.547,E2 -7646.547} C_VEL
LIN {X 0,Y 466.733,Z 859.271,A -85,B 0,C 180,E1 -7647.41,E2 -7647.41} C_VEL
LIN {X 0,Y 466.729,Z 860.276,A -85,B 0,C 180,E1 -7648.274,E2 -7648.274} C_VEL
LIN {X 0,Y 466.709,Z 860.897,A -85,B 0,C 180,E1 -7649.137,E2 -7649.137} C_VEL
LIN {X 0,Y 466.689,Z 861.114,A -85,B 0,C 180,E1 -7650,E2 -7650} C_VEL
LIN {X 0,Y 466.704,Z 860.891,A -85,B 0,C 180,E1 -7650.862,E2 -7650.862} C_VEL
LIN {X 0,Y 466.733,Z 859.245,A -85,B 0,C 180,E1 -7652.589,E2 -7652.589} C_VEL
LIN {X 0,Y 466.788,Z 857.797,A -85,B 0,C 180,E1 -7653.452,E2 -7653.452} C_VEL
LIN {X 0,Y 466.776,Z 854.786,A -85,B 0,C 180,E1 -7654.75,E2 -7654.75} C_VEL
LIN {X 0,Y 466.87,Z 850.701,A -85,B 0,C 180,E1 -7656.048,E2 -7656.048} C_VEL
LIN {X 0,Y 467.004,Z 844.392,A -85,B 0,C 180,E1 -7657.566,E2 -7657.566} C_VEL
LIN {X 0,Y 467.255,Z 837.506,A -85,B 0,C 180,E1 -7658.868,E2 -7658.868} C_VEL
LIN {X 0,Y 467.548,Z 828.883,A -85,B 0,C 180,E1 -7660.172,E2 -7660.172} C_VEL
LIN {X 0,Y 467.952,Z 819.976,A -85,B 0,C 180,E1 -7661.258,E2 -7661.258} C_VEL
LIN {X 0,Y 468.415,Z 809.525,A -85,B 0,C 180,E1 -7662.295,E2 -7662.295} C_VEL
LIN {X 0,Y 468.875,Z 796.479,A -85,B 0,C 180,E1 -7663.323,E2 -7663.323} C_VEL
LIN {X 0,Y 469.415,Z 784.474,A -85,B 0,C 180,E1 -7664.08,E2 -7664.08} C_VEL
LIN {X 0,Y 469.876,Z 772.047,A -85,B 0,C 180,E1 -7664.674,E2 -7664.674} C_VEL
LIN {X 0,Y 468.999,Z 763.252,A -85,B 0,C 180,E1 -7665.022,E2 -7665.022} C_VEL
LIN {X 0,Y 467.551,Z 749.707,A -85,B 0,C 180,E1 -7665.404,E2 -7665.404} C_VEL
LIN {X 0,Y 467.435,Z 747.874,A -85,B 0,C 180,E1 -7665.478,E2 -7665.478} C_VEL
LIN {X 0,Y 467.803,Z 732.034,A -85,B 0,C 180,E1 -7669.006,E2 -7669.006} C_VEL
LIN {X 0,Y 468.142,Z 717.517,A -85,B 0,C 180,E1 -7672.275,E2 -7672.275} C_VEL
LIN {X 0,Y 468.61,Z 704.317,A -85,B 0,C 180,E1 -7675.304,E2 -7675.304} C_VEL
LIN {X 0,Y 469.154,Z 690.084,A -85,B 0,C 180,E1 -7678.643,E2 -7678.643} C_VEL
LIN {X 0,Y 469.777,Z 675.877,A -85,B 0,C 180,E1 -7682.078,E2 -7682.078} C_VEL
LIN {X 0,Y 470.371,Z 663.662,A -85,B 0,C 180,E1 -7685.128,E2 -7685.128} C_VEL
LIN {X 0,Y 470.592,Z 657.646,A -85,B 0,C 180,E1 -7686.681,E2 -7686.681} C_VEL
LIN {X 0,Y 469.014,Z 649.357,A -85,B 0,C 180,E1 -7689.002,E2 -7689.002} C_VEL
LIN {X 0,Y 467.596,Z 642.242,A -85,B 0,C 180,E1 -7691.111,E2 -7691.111} C_VEL
LIN {X 0,Y 467.552,Z 642.244,A -85,B 0,C 180,E1 -7693.82,E2 -7693.82} C_VEL
LIN {X 0,Y 467.575,Z 642.244,A -85,B 0,C 180,E1 -7696.258,E2 -7696.258} C_VEL
LIN {X 0,Y 467.587,Z 642.242,A -85,B 0,C 180,E1 -7698.721,E2 -7698.721} C_VEL
LIN {X 0,Y 467.575,Z 642.239,A -85,B 0,C 180,E1 -7701.406,E2 -7701.406} C_VEL
LIN {X 0,Y 467.559,Z 642.245,A -85,B 0,C 180,E1 -7704.26,E2 -7704.26} C_VEL
LIN {X 0,Y 467.578,Z 642.24,A -85,B 0,C 180,E1 -7707.32,E2 -7707.32} C_VEL
LIN {X 0,Y 467.574,Z 642.238,A -85,B 0,C 180,E1 -7710.665,E2 -7710.665} C_VEL
LIN {X 0,Y 467.624,Z 642.236,A -85,B 0,C 180,E1 -7713.2,E2 -7713.2} C_VEL
LIN {X 0,Y 467.588,Z 642.237,A -85,B 0,C 180,E1 -7716.468,E2 -7716.468} C_VEL
LIN {X 0,Y 467.619,Z 642.234,A -85,B 0,C 180,E1 -7719.777,E2 -7719.777} C_VEL
LIN {X 0,Y 467.604,Z 642.235,A -85,B 0,C 180,E1 -7722.506,E2 -7722.506} C_VEL
LIN {X 0,Y 467.602,Z 642.24,A -85,B 0,C 180,E1 -7725.196,E2 -7725.196} C_VEL
LIN {X 0,Y 467.692,Z 642.225,A -85,B 0,C 180,E1 -7727.855,E2 -7727.855} C_VEL
LIN {X 0,Y 467.678,Z 642.229,A -85,B 0,C 180,E1 -7731.357,E2 -7731.357} C_VEL
LIN {X 0,Y 467.738,Z 642.222,A -85,B 0,C 180,E1 -7733.962,E2 -7733.962} C_VEL
LIN {X 0,Y 467.855,Z 642.206,A -85,B 0,C 180,E1 -7737.417,E2 -7737.417} C_VEL
LIN {X 0,Y 467.877,Z 642.209,A -85,B 0,C 180,E1 -7740,E2 -7740} C_VEL
LIN {X 0,Y 467.73,Z 642.226,A -85,B 0,C 180,E1 -7743.014,E2 -7743.014} C_VEL
LIN {X 0,Y 467.778,Z 642.768,A -85,B 0,C 180,E1 -7743.23,E2 -7743.23} C_VEL
LIN {X 0,Y 468.818,Z 650.167,A -85,B 0,C 180,E1 -7745.16,E2 -7745.16} C_VEL
LIN {X 0,Y 468.899,Z 662.882,A -85,B 0,C 180,E1 -7748.424,E2 -7748.424} C_VEL
LIN {X 0,Y 468.702,Z 675.345,A -85,B 0,C 180,E1 -7751.679,E2 -7751.679} C_VEL
LIN {X 0,Y 468.483,Z 686.958,A -85,B 0,C 180,E1 -7754.775,E2 -7754.775} C_VEL
LIN {X 0,Y 468.208,Z 698.569,A -85,B 0,C 180,E1 -7757.921,E2 -7757.921} C_VEL
LIN {X 0,Y 467.943,Z 710.448,A -85,B 0,C 180,E1 -7761.128,E2 -7761.128} C_VEL
LIN {X 0,Y 467.703,Z 722.403,A -85,B 0,C 180,E1 -7764.408,E2 -7764.408} C_VEL
LIN {X 0,Y 467.57,Z 726.851,A -85,B 0,C 180,E1 -7765.633,E2 -7765.633} C_VEL
LIN {X 0,Y 470.011,Z 740.947,A -85,B 0,C 180,E1 -7766.085,E2 -7766.085} C_VEL
LIN {X 0,Y 470.229,Z 745.891,A -85,B 0,C 180,E1 -7766.267,E2 -7766.267} C_VEL
LIN {X 0,Y 469.812,Z 758.809,A -85,B 0,C 180,E1 -7766.845,E2 -7766.845} C_VEL
LIN {X 0,Y 469.318,Z 770.412,A -85,B 0,C 180,E1 -7767.539,E2 -7767.539} C_VEL
LIN {X 0,Y 468.797,Z 782.194,A -85,B 0,C 180,E1 -7768.456,E2 -7768.456} C_VEL
LIN {X 0,Y 468.264,Z 792.762,A -85,B 0,C 180,E1 -7769.485,E2 -7769.485} C_VEL
LIN {X 0,Y 467.817,Z 802.781,A -85,B 0,C 180,E1 -7770.716,E2 -7770.716} C_VEL
LIN {X 0,Y 467.434,Z 810.998,A -85,B 0,C 180,E1 -7771.965,E2 -7771.965} C_VEL
LIN {X 0,Y 467.144,Z 818.079,A -85,B 0,C 180,E1 -7773.307,E2 -7773.307} C_VEL
LIN {X 0,Y 466.921,Z 823.073,A -85,B 0,C 180,E1 -7774.48,E2 -7774.48} C_VEL
LIN {X 0,Y 466.74,Z 827.961,A -85,B 0,C 180,E1 -7775.962,E2 -7775.962} C_VEL
LIN {X 0,Y 466.624,Z 831.785,A -85,B 0,C 180,E1 -7777.588,E2 -7777.588} C_VEL
LIN {X 0,Y 466.499,Z 834.105,A -85,B 0,C 180,E1 -7779.253,E2 -7779.253} C_VEL
LIN {X 0,Y 466.483,Z 834.859,A -85,B 0,C 180,E1 -7780.379,E2 -7780.379} C_VEL
LIN {X 0,Y 466.463,Z 834.891,A -85,B 0,C 180,E1 -7781.524,E2 -7781.524} C_VEL
LIN {X 0,Y 466.502,Z 834.229,A -85,B 0,C 180,E1 -7782.683,E2 -7782.683} C_VEL
LIN {X 0,Y 466.542,Z 832.832,A -85,B 0,C 180,E1 -7783.864,E2 -7783.864} C_VEL
LIN {X 0,Y 466.641,Z 830.618,A -85,B 0,C 180,E1 -7785.061,E2 -7785.061} C_VEL
LIN {X 0,Y 466.785,Z 827.489,A -85,B 0,C 180,E1 -7786.277,E2 -7786.277} C_VEL
LIN {X 0,Y 466.955,Z 822.342,A -85,B 0,C 180,E1 -7787.78,E2 -7787.78} C_VEL
LIN {X 0,Y 467.203,Z 815.694,A -85,B 0,C 180,E1 -7789.253,E2 -7789.253} C_VEL
LIN {X 0,Y 467.498,Z 808.841,A -85,B 0,C 180,E1 -7790.467,E2 -7790.467} C_VEL
LIN {X 0,Y 467.873,Z 800.372,A -85,B 0,C 180,E1 -7791.686,E2 -7791.686} C_VEL
LIN {X 0,Y 468.352,Z 791.153,A -85,B 0,C 180,E1 -7792.762,E2 -7792.762} C_VEL
LIN {X 0,Y 468.842,Z 780.939,A -85,B 0,C 180,E1 -7793.734,E2 -7793.734} C_VEL
LIN {X 0,Y 469.324,Z 769.628,A -85,B 0,C 180,E1 -7794.597,E2 -7794.597} C_VEL
LIN {X 0,Y 469.882,Z 757.492,A -85,B 0,C 180,E1 -7795.306,E2 -7795.306} C_VEL
LIN {X 0,Y 470.257,Z 745.182,A -85,B 0,C 180,E1 -7795.846,E2 -7795.846} C_VEL
LIN {X 0,Y 469.645,Z 738.667,A -85,B 0,C 180,E1 -7796.089,E2 -7796.089} C_VEL
LIN {X 0,Y 467.523,Z 726.644,A -85,B 0,C 180,E1 -7796.466,E2 -7796.466} C_VEL
LIN {X 0,Y 467.765,Z 716.828,A -85,B 0,C 180,E1 -7799.193,E2 -7799.193} C_VEL
LIN {X 0,Y 467.167,Z 714.557,A -85,B 0,C 180,E1 -7799.856,E2 -7799.856} C_VEL
LIN {X 0,Y 464.415,Z 711.073,A -85,B 0,C 180,E1 -7800.949,E2 -7800.949} C_VEL
LIN {X 0,Y 462.099,Z 708.313,A -85,B 0,C 180,E1 -7801.83,E2 -7801.83} C_VEL
LIN {X 0,Y 461.157,Z 706.083,A -85,B 0,C 180,E1 -7802.504,E2 -7802.504} C_VEL
LIN {X 0,Y 461.109,Z 705.291,A -85,B 0,C 180,E1 -7802.73,E2 -7802.73} C_VEL
LIN {X 0,Y 461.437,Z 694.616,A -85,B 0,C 180,E1 -7805.719,E2 -7805.719} C_VEL
LIN {X 0,Y 461.751,Z 682.763,A -85,B 0,C 180,E1 -7809.043,E2 -7809.043} C_VEL
LIN {X 0,Y 462.005,Z 672.817,A -85,B 0,C 180,E1 -7811.83,E2 -7811.83} C_VEL
LIN {X 0,Y 462.262,Z 661.38,A -85,B 0,C 180,E1 -7815.022,E2 -7815.022} C_VEL
LIN {X 0,Y 462.256,Z 653.404,A -85,B 0,C 180,E1 -7817.265,E2 -7817.265} C_VEL
LIN {X 0,Y 461.433,Z 647.333,A -85,B 0,C 180,E1 -7819.025,E2 -7819.025} C_VEL
LIN {X 0,Y 460.611,Z 643.112,A -85,B 0,C 180,E1 -7820.283,E2 -7820.283} C_VEL
LIN {X 0,Y 460.667,Z 643.106,A -85,B 0,C 180,E1 -7822.99,E2 -7822.99} C_VEL
LIN {X 0,Y 460.7,Z 643.102,A -85,B 0,C 180,E1 -7824.749,E2 -7824.749} C_VEL
LIN {X 0,Y 460.827,Z 643.086,A -85,B 0,C 180,E1 -7827.378,E2 -7827.378} C_VEL
LIN {X 0,Y 460.855,Z 643.08,A -85,B 0,C 180,E1 -7830,E2 -7830} C_VEL
LIN {X 0,Y 460.827,Z 643.083,A -85,B 0,C 180,E1 -7832.623,E2 -7832.623} C_VEL
LIN {X 0,Y 460.703,Z 643.098,A -85,B 0,C 180,E1 -7836.13,E2 -7836.13} C_VEL
LIN {X 0,Y 460.631,Z 643.109,A -85,B 0,C 180,E1 -7838.776,E2 -7838.776} C_VEL
LIN {X 0,Y 460.636,Z 643.108,A -85,B 0,C 180,E1 -7842.457,E2 -7842.457} C_VEL
LIN {X 0,Y 460.602,Z 643.111,A -85,B 0,C 180,E1 -7845.998,E2 -7845.998} C_VEL
LIN {X 0,Y 460.573,Z 643.117,A -85,B 0,C 180,E1 -7848.902,E2 -7848.902} C_VEL
LIN {X 0,Y 460.517,Z 643.123,A -85,B 0,C 180,E1 -7851.486,E2 -7851.486} C_VEL
LIN {X 0,Y 460.579,Z 643.284,A -85,B 0,C 180,E1 -7853.226,E2 -7853.226} C_VEL
LIN {X 0,Y 463.511,Z 654.034,A -85,B 0,C 180,E1 -7853.911,E2 -7853.911} C_VEL
LIN {X 0,Y 463.186,Z 666.186,A -85,B 0,C 180,E1 -7854.748,E2 -7854.748} C_VEL
LIN {X 0,Y 462.701,Z 676.633,A -85,B 0,C 180,E1 -7855.651,E2 -7855.651} C_VEL
LIN {X 0,Y 462.282,Z 686.068,A -85,B 0,C 180,E1 -7856.658,E2 -7856.658} C_VEL
LIN {X 0,Y 461.822,Z 695.639,A -85,B 0,C 180,E1 -7857.927,E2 -7857.927} C_VEL
LIN {X 0,Y 461.403,Z 703.23,A -85,B 0,C 180,E1 -7859.171,E2 -7859.171} C_VEL
LIN {X 0,Y 461.081,Z 709.565,A -85,B 0,C 180,E1 -7860.452,E2 -7860.452} C_VEL
LIN {X 0,Y 460.806,Z 714.768,A -85,B 0,C 180,E1 -7861.766,E2 -7861.766} C_VEL
LIN {X 0,Y 460.563,Z 719.456,A -85,B 0,C 180,E1 -7863.322,E2 -7863.322} C_VEL
LIN {X 0,Y 460.417,Z 722.036,A -85,B 0,C 180,E1 -7864.485,E2 -7864.485} C_VEL
LIN {X 0,Y 460.281,Z 724.266,A -85,B 0,C 180,E1 -7865.977,E2 -7865.977} C_VEL
LIN {X 0,Y 460.254,Z 725.365,A -85,B 0,C 180,E1 -7867.647,E2 -7867.647} C_VEL
LIN {X 0,Y 460.294,Z 725.307,A -85,B 0,C 180,E1 -7868.859,E2 -7868.859} C_VEL
LIN {X 0,Y 460.367,Z 724.32,A -85,B 0,C 180,E1 -7870.244,E2 -7870.244} C_VEL
LIN {X 0,Y 460.455,Z 722.415,A -85,B 0,C 180,E1 -7871.592,E2 -7871.592} C_VEL
LIN {X 0,Y 460.662,Z 719.556,A -85,B 0,C 180,E1 -7872.92,E2 -7872.92} C_VEL
LIN {X 0,Y 460.938,Z 714.644,A -85,B 0,C 180,E1 -7874.537,E2 -7874.537} C_VEL
LIN {X 0,Y 461.301,Z 708.796,A -85,B 0,C 180,E1 -7875.986,E2 -7875.986} C_VEL
LIN {X 0,Y 461.599,Z 702.603,A -85,B 0,C 180,E1 -7877.207,E2 -7877.207} C_VEL
LIN {X 0,Y 462.076,Z 694.775,A -85,B 0,C 180,E1 -7878.452,E2 -7878.452} C_VEL
LIN {X 0,Y 462.528,Z 685.326,A -85,B 0,C 180,E1 -7879.666,E2 -7879.666} C_VEL
LIN {X 0,Y 463.053,Z 675.128,A -85,B 0,C 180,E1 -7880.719,E2 -7880.719} C_VEL
LIN {X 0,Y 463.476,Z 663.956,A -85,B 0,C 180,E1 -7881.635,E2 -7881.635} C_VEL
LIN {X 0,Y 463.75,Z 654.774,A -85,B 0,C 180,E1 -7882.241,E2 -7882.241} C_VEL
LIN {X 0,Y 461.385,Z 646.112,A -85,B 0,C 180,E1 -7882.811,E2 -7882.811} C_VEL
LIN {X 0,Y 460.526,Z 643.122,A -85,B 0,C 180,E1 -7882.998,E2 -7882.998} C_VEL
LIN {X 0,Y 460.547,Z 643.121,A -85,B 0,C 180,E1 -7885.624,E2 -7885.624} C_VEL
LIN {X 0,Y 460.538,Z 643.117,A -85,B 0,C 180,E1 -7888.745,E2 -7888.745} C_VEL
LIN {X 0,Y 460.582,Z 643.112,A -85,B 0,C 180,E1 -7892.254,E2 -7892.254} C_VEL
LIN {X 0,Y 460.54,Z 643.114,A -85,B 0,C 180,E1 -7894.704,E2 -7894.704} C_VEL
LIN {X 0,Y 460.511,Z 643.118,A -85,B 0,C 180,E1 -7897.571,E2 -7897.571} C_VEL
LIN {X 0,Y 460.57,Z 643.113,A -85,B 0,C 180,E1 -7900.385,E2 -7900.385} C_VEL
LIN {X 0,Y 460.633,Z 643.109,A -85,B 0,C 180,E1 -7904.06,E2 -7904.06} C_VEL
LIN {X 0,Y 460.61,Z 643.111,A -85,B 0,C 180,E1 -7907.666,E2 -7907.666} C_VEL
LIN {X 0,Y 460.63,Z 643.103,A -85,B 0,C 180,E1 -7911.224,E2 -7911.224} C_VEL
LIN {X 0,Y 460.711,Z 643.096,A -85,B 0,C 180,E1 -7913.87,E2 -7913.87} C_VEL
LIN {X 0,Y 460.826,Z 643.075,A -85,B 0,C 180,E1 -7917.378,E2 -7917.378} C_VEL
LIN {X 0,Y 460.855,Z 643.079,A -85,B 0,C 180,E1 -7920,E2 -7920} C_VEL
LIN {X 0,Y 460.827,Z 643.08,A -85,B 0,C 180,E1 -7922.622,E2 -7922.622} C_VEL
LIN {X 0,Y 460.711,Z 643.096,A -85,B 0,C 180,E1 -7926.13,E2 -7926.13} C_VEL
LIN {X 0,Y 460.63,Z 643.1,A -85,B 0,C 180,E1 -7928.776,E2 -7928.776} C_VEL
LIN {X 0,Y 460.615,Z 643.106,A -85,B 0,C 180,E1 -7932.445,E2 -7932.445} C_VEL
LIN {X 0,Y 460.602,Z 643.111,A -85,B 0,C 180,E1 -7935.998,E2 -7935.998} C_VEL
LIN {X 0,Y 460.572,Z 643.11,A -85,B 0,C 180,E1 -7938.902,E2 -7938.902} C_VEL
LIN {X 0,Y 460.517,Z 643.117,A -85,B 0,C 180,E1 -7941.486,E2 -7941.486} C_VEL
LIN {X 0,Y 460.543,Z 643.12,A -85,B 0,C 180,E1 -7944.332,E2 -7944.332} C_VEL
LIN {X 0,Y 460.575,Z 643.111,A -85,B 0,C 180,E1 -7947.244,E2 -7947.244} C_VEL
LIN {X 0,Y 460.512,Z 643.123,A -85,B 0,C 180,E1 -7950.24,E2 -7950.24} C_VEL
LIN {X 0,Y 460.531,Z 643.118,A -85,B 0,C 180,E1 -7953.325,E2 -7953.325} C_VEL
LIN {X 0,Y 460.478,Z 643.129,A -85,B 0,C 180,E1 -7956.53,E2 -7956.53} C_VEL
LIN {X 0,Y 460.535,Z 643.118,A -85,B 0,C 180,E1 -7959.862,E2 -7959.862} C_VEL
LIN {X 0,Y 460.515,Z 643.119,A -85,B 0,C 180,E1 -7962.9,E2 -7962.9} C_VEL
LIN {X 0,Y 460.514,Z 643.122,A -85,B 0,C 180,E1 -7965.83,E2 -7965.83} C_VEL
LIN {X 0,Y 460.577,Z 643.253,A -85,B 0,C 180,E1 -7969.236,E2 -7969.236} C_VEL
LIN {X 0,Y 462.542,Z 653.189,A -85,B 0,C 180,E1 -7972.195,E2 -7972.195} C_VEL
LIN {X 0,Y 463.245,Z 658.643,A -85,B 0,C 180,E1 -7973.724,E2 -7973.724} C_VEL
LIN {X 0,Y 462.564,Z 671.803,A -85,B 0,C 180,E1 -7977.1,E2 -7977.1} C_VEL
LIN {X 0,Y 462.058,Z 684.018,A -85,B 0,C 180,E1 -7980.11,E2 -7980.11} C_VEL
LIN {X 0,Y 461.583,Z 698.476,A -85,B 0,C 180,E1 -7983.554,E2 -7983.554} C_VEL
LIN {X 0,Y 461.158,Z 711.914,A -85,B 0,C 180,E1 -7986.657,E2 -7986.657} C_VEL
LIN {X 0,Y 460.748,Z 726.352,A -85,B 0,C 180,E1 -7989.928,E2 -7989.928} C_VEL
LIN {X 0,Y 460.472,Z 739.751,A -85,B 0,C 180,E1 -7992.914,E2 -7992.914} C_VEL
LIN {X 0,Y 460.37,Z 746.057,A -85,B 0,C 180,E1 -7994.313,E2 -7994.313} C_VEL
LIN {X 0,Y 461.68,Z 760.875,A -85,B 0,C 180,E1 -7994.722,E2 -7994.722} C_VEL
LIN {X 0,Y 462.878,Z 771.443,A -85,B 0,C 180,E1 -7995.154,E2 -7995.154} C_VEL
LIN {X 0,Y 462.256,Z 789.209,A -85,B 0,C 180,E1 -7996.033,E2 -7996.033} C_VEL
LIN {X 0,Y 461.787,Z 800.835,A -85,B 0,C 180,E1 -7996.803,E2 -7996.803} C_VEL
LIN {X 0,Y 461.299,Z 812.471,A -85,B 0,C 180,E1 -7997.796,E2 -7997.796} C_VEL
LIN {X 0,Y 460.87,Z 821.846,A -85,B 0,C 180,E1 -7998.788,E2 -7998.788} C_VEL
LIN {X 0,Y 460.473,Z 830.368,A -85,B 0,C 180,E1 -7999.891,E2 -7999.891} C_VEL
LIN {X 0,Y 460.165,Z 838.641,A -85,B 0,C 180,E1 -8001.215,E2 -8001.215} C_VEL
LIN {X 0,Y 459.902,Z 845.281,A -85,B 0,C 180,E1 -8002.536,E2 -8002.536} C_VEL
LIN {X 0,Y 459.796,Z 850.556,A -85,B 0,C 180,E1 -8003.857,E2 -8003.857} C_VEL
LIN {X 0,Y 459.704,Z 854.631,A -85,B 0,C 180,E1 -8005.176,E2 -8005.176} C_VEL
LIN {X 0,Y 459.689,Z 857.629,A -85,B 0,C 180,E1 -8006.493,E2 -8006.493} C_VEL
LIN {X 0,Y 459.654,Z 859.07,A -85,B 0,C 180,E1 -8007.371,E2 -8007.371} C_VEL
LIN {X 0,Y 459.634,Z 860.081,A -85,B 0,C 180,E1 -8008.247,E2 -8008.247} C_VEL
LIN {X 0,Y 459.637,Z 860.698,A -85,B 0,C 180,E1 -8009.123,E2 -8009.123} C_VEL
LIN {X 0,Y 459.615,Z 860.916,A -85,B 0,C 180,E1 -8010,E2 -8010} C_VEL
LIN {X 0,Y 459.632,Z 860.689,A -85,B 0,C 180,E1 -8010.876,E2 -8010.876} C_VEL
LIN {X 0,Y 459.631,Z 860.062,A -85,B 0,C 180,E1 -8011.752,E2 -8011.752} C_VEL
LIN {X 0,Y 459.653,Z 859.04,A -85,B 0,C 180,E1 -8012.629,E2 -8012.629} C_VEL
LIN {X 0,Y 459.684,Z 857.59,A -85,B 0,C 180,E1 -8013.506,E2 -8013.506} C_VEL
LIN {X 0,Y 459.7,Z 854.576,A -85,B 0,C 180,E1 -8014.823,E2 -8014.823} C_VEL
LIN {X 0,Y 459.778,Z 850.485,A -85,B 0,C 180,E1 -8016.142,E2 -8016.142} C_VEL
LIN {X 0,Y 459.927,Z 844.169,A -85,B 0,C 180,E1 -8017.683,E2 -8017.683} C_VEL
LIN {X 0,Y 460.176,Z 837.276,A -85,B 0,C 180,E1 -8019.006,E2 -8019.006} C_VEL
LIN {X 0,Y 460.455,Z 830.227,A -85,B 0,C 180,E1 -8020.109,E2 -8020.109} C_VEL
LIN {X 0,Y 460.861,Z 821.691,A -85,B 0,C 180,E1 -8021.211,E2 -8021.211} C_VEL
LIN {X 0,Y 461.347,Z 811.115,A -85,B 0,C 180,E1 -8022.314,E2 -8022.314} C_VEL
LIN {X 0,Y 461.741,Z 800.621,A -85,B 0,C 180,E1 -8023.197,E2 -8023.197} C_VEL
LIN {X 0,Y 462.297,Z 787.268,A -85,B 0,C 180,E1 -8024.077,E2 -8024.077} C_VEL
LIN {X 0,Y 462.808,Z 774.89,A -85,B 0,C 180,E1 -8024.735,E2 -8024.735} C_VEL
LIN {X 0,Y 462.802,Z 769.714,A -85,B 0,C 180,E1 -8024.96,E2 -8024.96} C_VEL
LIN {X 0,Y 461.357,Z 757.077,A -85,B 0,C 180,E1 -8025.429,E2 -8025.429} C_VEL
LIN {X 0,Y 460.387,Z 747.121,A -85,B 0,C 180,E1 -8025.687,E2 -8025.687} C_VEL
LIN {X 0,Y 460.729,Z 731.484,A -85,B 0,C 180,E1 -8029.223,E2 -8029.223} C_VEL
LIN {X 0,Y 461.111,Z 717.682,A -85,B 0,C 180,E1 -8032.397,E2 -8032.397} C_VEL
LIN {X 0,Y 461.545,Z 705.52,A -85,B 0,C 180,E1 -8035.236,E2 -8035.236} C_VEL
LIN {X 0,Y 462.137,Z 691.344,A -85,B 0,C 180,E1 -8038.622,E2 -8038.622} C_VEL
LIN {X 0,Y 462.7,Z 678.69,A -85,B 0,C 180,E1 -8041.724,E2 -8041.724} C_VEL
LIN {X 0,Y 463.313,Z 667.394,A -85,B 0,C 180,E1 -8044.581,E2 -8044.581} C_VEL
LIN {X 0,Y 463.67,Z 659.793,A -85,B 0,C 180,E1 -8046.55,E2 -8046.55} C_VEL
LIN {X 0,Y 462.767,Z 654.112,A -85,B 0,C 180,E1 -8048.142,E2 -8048.142} C_VEL
LIN {X 0,Y 460.542,Z 643.12,A -85,B 0,C 180,E1 -8051.397,E2 -8051.397} C_VEL
LIN {X 0,Y 460.514,Z 643.124,A -85,B 0,C 180,E1 -8054.588,E2 -8054.588} C_VEL
LIN {X 0,Y 460.545,Z 643.117,A -85,B 0,C 180,E1 -8057.821,E2 -8057.821} C_VEL
LIN {X 0,Y 460.566,Z 643.113,A -85,B 0,C 180,E1 -8061.098,E2 -8061.098} C_VEL
LIN {X 0,Y 460.509,Z 643.119,A -85,B 0,C 180,E1 -8064.554,E2 -8064.554} C_VEL
LIN {X 0,Y 460.528,Z 643.121,A -85,B 0,C 180,E1 -8067.715,E2 -8067.715} C_VEL
LIN {X 0,Y 460.543,Z 643.114,A -85,B 0,C 180,E1 -8070.769,E2 -8070.769} C_VEL
LIN {X 0,Y 460.564,Z 643.114,A -85,B 0,C 180,E1 -8073.735,E2 -8073.735} C_VEL
LIN {X 0,Y 460.542,Z 643.115,A -85,B 0,C 180,E1 -8076.624,E2 -8076.624} C_VEL
LIN {X 0,Y 460.547,Z 643.117,A -85,B 0,C 180,E1 -8079.452,E2 -8079.452} C_VEL
LIN {X 0,Y 460.554,Z 643.112,A -85,B 0,C 180,E1 -8082.23,E2 -8082.23} C_VEL
LIN {X 0,Y 460.561,Z 643.116,A -85,B 0,C 180,E1 -8084.965,E2 -8084.965} C_VEL
LIN {X 0,Y 460.652,Z 643.103,A -85,B 0,C 180,E1 -8087.667,E2 -8087.667} C_VEL
LIN {X 0,Y 460.625,Z 643.108,A -85,B 0,C 180,E1 -8091.224,E2 -8091.224} C_VEL
LIN {X 0,Y 460.704,Z 643.098,A -85,B 0,C 180,E1 -8093.87,E2 -8093.87} C_VEL
LIN {X 0,Y 460.82,Z 643.083,A -85,B 0,C 180,E1 -8097.377,E2 -8097.377} C_VEL
LIN {X 0,Y 460.847,Z 643.084,A -85,B 0,C 180,E1 -8100,E2 -8100} C_VEL
LIN {X 0,Y 460.754,Z 643.159,A -85,B 0,C 180,E1 -8102.869,E2 -8102.869} C_VEL
LIN {X 0,Y 461.787,Z 650.473,A -85,B 0,C 180,E1 -8104.801,E2 -8104.801} C_VEL
LIN {X 0,Y 461.918,Z 658.95,A -85,B 0,C 180,E1 -8106.991,E2 -8106.991} C_VEL
LIN {X 0,Y 461.85,Z 669.08,A -85,B 0,C 180,E1 -8109.636,E2 -8109.636} C_VEL
LIN {X 0,Y 461.675,Z 680.352,A -85,B 0,C 180,E1 -8112.651,E2 -8112.651} C_VEL
LIN {X 0,Y 461.376,Z 692.544,A -85,B 0,C 180,E1 -8115.914,E2 -8115.914} C_VEL
LIN {X 0,Y 461.135,Z 702.633,A -85,B 0,C 180,E1 -8118.666,E2 -8118.666} C_VEL
LIN {X 0,Y 460.913,Z 713.127,A -85,B 0,C 180,E1 -8121.548,E2 -8121.548} C_VEL
LIN {X 0,Y 460.687,Z 723.154,A -85,B 0,C 180,E1 -8124.324,E2 -8124.324} C_VEL
LIN {X 0,Y 460.568,Z 727.035,A -85,B 0,C 180,E1 -8125.399,E2 -8125.399} C_VEL
LIN {X 0,Y 463.02,Z 740.754,A -85,B 0,C 180,E1 -8125.842,E2 -8125.842} C_VEL
LIN {X 0,Y 463.384,Z 745.58,A -85,B 0,C 180,E1 -8126.025,E2 -8126.025} C_VEL
LIN {X 0,Y 462.944,Z 758.974,A -85,B 0,C 180,E1 -8126.63,E2 -8126.63} C_VEL
LIN {X 0,Y 462.382,Z 771.133,A -85,B 0,C 180,E1 -8127.373,E2 -8127.373} C_VEL
LIN {X 0,Y 461.856,Z 782.429,A -85,B 0,C 180,E1 -8128.27,E2 -8128.27} C_VEL
LIN {X 0,Y 461.407,Z 791.627,A -85,B 0,C 180,E1 -8129.171,E2 -8129.171} C_VEL
LIN {X 0,Y 460.941,Z 800.387,A -85,B 0,C 180,E1 -8130.209,E2 -8130.209} C_VEL
LIN {X 0,Y 460.488,Z 809.316,A -85,B 0,C 180,E1 -8131.515,E2 -8131.515} C_VEL
LIN {X 0,Y 460.147,Z 816.679,A -85,B 0,C 180,E1 -8132.858,E2 -8132.858} C_VEL
LIN {X 0,Y 459.92,Z 822.274,A -85,B 0,C 180,E1 -8134.127,E2 -8134.127} C_VEL
LIN {X 0,Y 459.733,Z 827.101,A -85,B 0,C 180,E1 -8135.515,E2 -8135.515} C_VEL
LIN {X 0,Y 459.61,Z 830.022,A -85,B 0,C 180,E1 -8136.609,E2 -8136.609} C_VEL
LIN {X 0,Y 459.528,Z 832.301,A -85,B 0,C 180,E1 -8137.717,E2 -8137.717} C_VEL
LIN {X 0,Y 459.44,Z 833.917,A -85,B 0,C 180,E1 -8138.842,E2 -8138.842} C_VEL
LIN {X 0,Y 459.403,Z 834.926,A -85,B 0,C 180,E1 -8140.103,E2 -8140.103} C_VEL
LIN {X 0,Y 459.362,Z 835.107,A -85,B 0,C 180,E1 -8141.439,E2 -8141.439} C_VEL
LIN {X 0,Y 459.416,Z 834.384,A -85,B 0,C 180,E1 -8142.754,E2 -8142.754} C_VEL
LIN {X 0,Y 459.46,Z 832.816,A -85,B 0,C 180,E1 -8144.036,E2 -8144.036} C_VEL
LIN {X 0,Y 459.561,Z 830.416,A -85,B 0,C 180,E1 -8145.295,E2 -8145.295} C_VEL
LIN {X 0,Y 459.736,Z 826.021,A -85,B 0,C 180,E1 -8146.896,E2 -8146.896} C_VEL
LIN {X 0,Y 459.883,Z 821.476,A -85,B 0,C 180,E1 -8148.143,E2 -8148.143} C_VEL
LIN {X 0,Y 460.167,Z 815.794,A -85,B 0,C 180,E1 -8149.394,E2 -8149.394} C_VEL
LIN {X 0,Y 460.511,Z 808.81,A -85,B 0,C 180,E1 -8150.643,E2 -8150.643} C_VEL
LIN {X 0,Y 460.898,Z 800.412,A -85,B 0,C 180,E1 -8151.863,E2 -8151.863} C_VEL
LIN {X 0,Y 461.423,Z 790.6,A -85,B 0,C 180,E1 -8153.014,E2 -8153.014} C_VEL
LIN {X 0,Y 461.979,Z 779.602,A -85,B 0,C 180,E1 -8154.056,E2 -8154.056} C_VEL
LIN {X 0,Y 462.455,Z 769.228,A -85,B 0,C 180,E1 -8154.836,E2 -8154.836} C_VEL
LIN {X 0,Y 463.034,Z 756.349,A -85,B 0,C 180,E1 -8155.587,E2 -8155.587} C_VEL
LIN {X 0,Y 463.393,Z 743.728,A -85,B 0,C 180,E1 -8156.127,E2 -8156.127} C_VEL
LIN {X 0,Y 461.269,Z 730.874,A -85,B 0,C 180,E1 -8156.573,E2 -8156.573} C_VEL
LIN {X 0,Y 460.525,Z 726.768,A -85,B 0,C 180,E1 -8156.705,E2 -8156.705} C_VEL
LIN {X 0,Y 460.823,Z 714.606,A -85,B 0,C 180,E1 -8160.118,E2 -8160.118} C_VEL
LIN {X 0,Y 461.109,Z 705.291,A -85,B 0,C 180,E1 -8162.73,E2 -8162.73} C_VEL
LIN {X 0,Y 460.545,Z 703.002,A -85,B 0,C 180,E1 -8163.403,E2 -8163.403} C_VEL
LIN {X 0,Y 457.83,Z 699.549,A -85,B 0,C 180,E1 -8164.512,E2 -8164.512} C_VEL
LIN {X 0,Y 455.514,Z 696.803,A -85,B 0,C 180,E1 -8165.407,E2 -8165.407} C_VEL
LIN {X 0,Y 454.547,Z 694.565,A -85,B 0,C 180,E1 -8166.09,E2 -8166.09} C_VEL
LIN {X 0,Y 454.485,Z 693.766,A -85,B 0,C 180,E1 -8166.318,E2 -8166.318} C_VEL
LIN {X 0,Y 454.852,Z 681.928,A -85,B 0,C 180,E1 -8169.657,E2 -8169.657} C_VEL
LIN {X 0,Y 455.121,Z 670.326,A -85,B 0,C 180,E1 -8172.939,E2 -8172.939} C_VEL
LIN {X 0,Y 455.336,Z 660.523,A -85,B 0,C 180,E1 -8175.703,E2 -8175.703} C_VEL
LIN {X 0,Y 455.267,Z 654.141,A -85,B 0,C 180,E1 -8177.519,E2 -8177.519} C_VEL
LIN {X 0,Y 454.06,Z 646.57,A -85,B 0,C 180,E1 -8179.747,E2 -8179.747} C_VEL
LIN {X 0,Y 453.584,Z 643.988,A -85,B 0,C 180,E1 -8180.525,E2 -8180.525} C_VEL
LIN {X 0,Y 453.631,Z 643.983,A -85,B 0,C 180,E1 -8182.881,E2 -8182.881} C_VEL
LIN {X 0,Y 453.673,Z 643.978,A -85,B 0,C 180,E1 -8184.667,E2 -8184.667} C_VEL
LIN {X 0,Y 453.767,Z 643.965,A -85,B 0,C 180,E1 -8187.337,E2 -8187.337} C_VEL
LIN {X 0,Y 453.826,Z 643.956,A -85,B 0,C 180,E1 -8190,E2 -8190} C_VEL
LIN {X 0,Y 453.767,Z 643.963,A -85,B 0,C 180,E1 -8192.664,E2 -8192.664} C_VEL
LIN {X 0,Y 453.671,Z 643.973,A -85,B 0,C 180,E1 -8196.226,E2 -8196.226} C_VEL
LIN {X 0,Y 453.595,Z 643.984,A -85,B 0,C 180,E1 -8198.914,E2 -8198.914} C_VEL
LIN {X 0,Y 453.604,Z 643.984,A -85,B 0,C 180,E1 -8202.551,E2 -8202.551} C_VEL
LIN {X 0,Y 453.547,Z 643.991,A -85,B 0,C 180,E1 -8206.196,E2 -8206.196} C_VEL
LIN {X 0,Y 453.522,Z 643.996,A -85,B 0,C 180,E1 -8209.041,E2 -8209.041} C_VEL
LIN {X 0,Y 453.478,Z 644.002,A -85,B 0,C 180,E1 -8211.836,E2 -8211.836} C_VEL
LIN {X 0,Y 453.5,Z 643.998,A -85,B 0,C 180,E1 -8212.976,E2 -8212.976} C_VEL
LIN {X 0,Y 456.638,Z 654.92,A -85,B 0,C 180,E1 -8213.697,E2 -8213.697} C_VEL
LIN {X 0,Y 456.379,Z 665.988,A -85,B 0,C 180,E1 -8214.461,E2 -8214.461} C_VEL
LIN {X 0,Y 455.839,Z 677.306,A -85,B 0,C 180,E1 -8215.441,E2 -8215.441} C_VEL
LIN {X 0,Y 455.387,Z 686.922,A -85,B 0,C 180,E1 -8216.477,E2 -8216.477} C_VEL
LIN {X 0,Y 454.981,Z 695.478,A -85,B 0,C 180,E1 -8217.607,E2 -8217.607} C_VEL
LIN {X 0,Y 454.492,Z 703.425,A -85,B 0,C 180,E1 -8218.897,E2 -8218.897} C_VEL
LIN {X 0,Y 454.126,Z 710.296,A -85,B 0,C 180,E1 -8220.284,E2 -8220.284} C_VEL
LIN {X 0,Y 453.822,Z 716.105,A -85,B 0,C 180,E1 -8221.772,E2 -8221.772} C_VEL
LIN {X 0,Y 453.586,Z 720.342,A -85,B 0,C 180,E1 -8223.208,E2 -8223.208} C_VEL
LIN {X 0,Y 453.363,Z 723.593,A -85,B 0,C 180,E1 -8224.755,E2 -8224.755} C_VEL
LIN {X 0,Y 453.249,Z 725.571,A -85,B 0,C 180,E1 -8226.264,E2 -8226.264} C_VEL
LIN {X 0,Y 453.228,Z 726.407,A -85,B 0,C 180,E1 -8227.737,E2 -8227.737} C_VEL
LIN {X 0,Y 453.301,Z 726.049,A -85,B 0,C 180,E1 -8229.47,E2 -8229.47} C_VEL
LIN {X 0,Y 453.368,Z 724.953,A -85,B 0,C 180,E1 -8230.623,E2 -8230.623} C_VEL
LIN {X 0,Y 453.584,Z 721.952,A -85,B 0,C 180,E1 -8232.41,E2 -8232.41} C_VEL
LIN {X 0,Y 453.787,Z 718.768,A -85,B 0,C 180,E1 -8233.681,E2 -8233.681} C_VEL
LIN {X 0,Y 454.014,Z 714.628,A -85,B 0,C 180,E1 -8234.947,E2 -8234.947} C_VEL
LIN {X 0,Y 454.432,Z 708.463,A -85,B 0,C 180,E1 -8236.409,E2 -8236.409} C_VEL
LIN {X 0,Y 454.867,Z 700.633,A -85,B 0,C 180,E1 -8237.871,E2 -8237.871} C_VEL
LIN {X 0,Y 455.372,Z 692.111,A -85,B 0,C 180,E1 -8239.134,E2 -8239.134} C_VEL
LIN {X 0,Y 455.937,Z 682.359,A -85,B 0,C 180,E1 -8240.294,E2 -8240.294} C_VEL
LIN {X 0,Y 456.404,Z 671.605,A -85,B 0,C 180,E1 -8241.327,E2 -8241.327} C_VEL
LIN {X 0,Y 456.788,Z 660.462,A -85,B 0,C 180,E1 -8242.17,E2 -8242.17} C_VEL
LIN {X 0,Y 456.843,Z 655.332,A -85,B 0,C 180,E1 -8242.498,E2 -8242.498} C_VEL
LIN {X 0,Y 453.502,Z 643.996,A -85,B 0,C 180,E1 -8243.248,E2 -8243.248} C_VEL
LIN {X 0,Y 453.477,Z 643.998,A -85,B 0,C 180,E1 -8246.087,E2 -8246.087} C_VEL
LIN {X 0,Y 453.477,Z 644,A -85,B 0,C 180,E1 -8249.241,E2 -8249.241} C_VEL
LIN {X 0,Y 453.537,Z 643.989,A -85,B 0,C 180,E1 -8252.298,E2 -8252.298} C_VEL
LIN {X 0,Y 453.501,Z 643.994,A -85,B 0,C 180,E1 -8255.265,E2 -8255.265} C_VEL
LIN {X 0,Y 453.481,Z 643.997,A -85,B 0,C 180,E1 -8258.415,E2 -8258.415} C_VEL
LIN {X 0,Y 453.523,Z 643.99,A -85,B 0,C 180,E1 -8261.009,E2 -8261.009} C_VEL
LIN {X 0,Y 453.577,Z 643.99,A -85,B 0,C 180,E1 -8263.877,E2 -8263.877} C_VEL
LIN {X 0,Y 453.565,Z 643.987,A -85,B 0,C 180,E1 -8267.471,E2 -8267.471} C_VEL
LIN {X 0,Y 453.593,Z 643.979,A -85,B 0,C 180,E1 -8271.087,E2 -8271.087} C_VEL
LIN {X 0,Y 453.678,Z 643.971,A -85,B 0,C 180,E1 -8273.775,E2 -8273.775} C_VEL
LIN {X 0,Y 453.767,Z 643.954,A -85,B 0,C 180,E1 -8277.337,E2 -8277.337} C_VEL
LIN {X 0,Y 453.825,Z 643.954,A -85,B 0,C 180,E1 -8280,E2 -8280} C_VEL
LIN {X 0,Y 453.767,Z 643.959,A -85,B 0,C 180,E1 -8282.663,E2 -8282.663} C_VEL
LIN {X 0,Y 453.679,Z 643.974,A -85,B 0,C 180,E1 -8286.225,E2 -8286.225} C_VEL
LIN {X 0,Y 453.594,Z 643.975,A -85,B 0,C 180,E1 -8288.913,E2 -8288.913} C_VEL
LIN {X 0,Y 453.565,Z 643.983,A -85,B 0,C 180,E1 -8292.529,E2 -8292.529} C_VEL
LIN {X 0,Y 453.546,Z 643.989,A -85,B 0,C 180,E1 -8296.196,E2 -8296.196} C_VEL
LIN {X 0,Y 453.521,Z 643.988,A -85,B 0,C 180,E1 -8299.041,E2 -8299.041} C_VEL
LIN {X 0,Y 453.478,Z 643.996,A -85,B 0,C 180,E1 -8301.836,E2 -8301.836} C_VEL
LIN {X 0,Y 453.515,Z 643.992,A -85,B 0,C 180,E1 -8304.735,E2 -8304.735} C_VEL
LIN {X 0,Y 453.534,Z 643.99,A -85,B 0,C 180,E1 -8307.96,E2 -8307.96} C_VEL
LIN {X 0,Y 453.467,Z 643.997,A -85,B 0,C 180,E1 -8311.525,E2 -8311.525} C_VEL
LIN {X 0,Y 453.489,Z 643.999,A -85,B 0,C 180,E1 -8314.777,E2 -8314.777} C_VEL
LIN {X 0,Y 453.467,Z 644.002,A -85,B 0,C 180,E1 -8318.312,E2 -8318.312} C_VEL
LIN {X 0,Y 453.496,Z 644,A -85,B 0,C 180,E1 -8320.609,E2 -8320.609} C_VEL
LIN {X 0,Y 453.458,Z 643.998,A -85,B 0,C 180,E1 -8323.244,E2 -8323.244} C_VEL
LIN {X 0,Y 453.469,Z 644,A -85,B 0,C 180,E1 -8325.779,E2 -8325.779} C_VEL
LIN {X 0,Y 453.51,Z 644.018,A -85,B 0,C 180,E1 -8328.887,E2 -8328.887} C_VEL
LIN {X 0,Y 455.456,Z 653.885,A -85,B 0,C 180,E1 -8331.903,E2 -8331.903} C_VEL
LIN {X 0,Y 456.203,Z 658.483,A -85,B 0,C 180,E1 -8333.234,E2 -8333.234} C_VEL
LIN {X 0,Y 456.011,Z 664.231,A -85,B 0,C 180,E1 -8334.769,E2 -8334.769} C_VEL
LIN {X 0,Y 455.422,Z 677.019,A -85,B 0,C 180,E1 -8338.077,E2 -8338.077} C_VEL
LIN {X 0,Y 454.808,Z 690.349,A -85,B 0,C 180,E1 -8341.377,E2 -8341.377} C_VEL
LIN {X 0,Y 454.352,Z 703.723,A -85,B 0,C 180,E1 -8344.58,E2 -8344.58} C_VEL
LIN {X 0,Y 453.91,Z 717.102,A -85,B 0,C 180,E1 -8347.707,E2 -8347.707} C_VEL
LIN {X 0,Y 453.576,Z 732.5,A -85,B 0,C 180,E1 -8351.245,E2 -8351.245} C_VEL
LIN {X 0,Y 453.275,Z 744.961,A -85,B 0,C 180,E1 -8354.06,E2 -8354.06} C_VEL
LIN {X 0,Y 454.602,Z 759.886,A -85,B 0,C 180,E1 -8354.481,E2 -8354.481} C_VEL
LIN {X 0,Y 455.882,Z 772.906,A -85,B 0,C 180,E1 -8355.035,E2 -8355.035} C_VEL
LIN {X 0,Y 455.516,Z 784.988,A -85,B 0,C 180,E1 -8355.594,E2 -8355.594} C_VEL
LIN {X 0,Y 454.932,Z 797.529,A -85,B 0,C 180,E1 -8356.373,E2 -8356.373} C_VEL
LIN {X 0,Y 454.507,Z 808.386,A -85,B 0,C 180,E1 -8357.243,E2 -8357.243} C_VEL
LIN {X 0,Y 454.055,Z 817.702,A -85,B 0,C 180,E1 -8358.165,E2 -8358.165} C_VEL
LIN {X 0,Y 453.572,Z 826.928,A -85,B 0,C 180,E1 -8359.284,E2 -8359.284} C_VEL
LIN {X 0,Y 453.199,Z 835.878,A -85,B 0,C 180,E1 -8360.628,E2 -8360.628} C_VEL
LIN {X 0,Y 452.919,Z 843.047,A -85,B 0,C 180,E1 -8361.972,E2 -8361.972} C_VEL
LIN {X 0,Y 452.732,Z 849.294,A -85,B 0,C 180,E1 -8363.469,E2 -8363.469} C_VEL
LIN {X 0,Y 452.635,Z 854.431,A -85,B 0,C 180,E1 -8365.101,E2 -8365.101} C_VEL
LIN {X 0,Y 452.586,Z 857.43,A -85,B 0,C 180,E1 -8366.438,E2 -8366.438} C_VEL
LIN {X 0,Y 452.576,Z 858.872,A -85,B 0,C 180,E1 -8367.329,E2 -8367.329} C_VEL
LIN {X 0,Y 452.567,Z 860.5,A -85,B 0,C 180,E1 -8369.11,E2 -8369.11} C_VEL
LIN {X 0,Y 452.544,Z 860.718,A -85,B 0,C 180,E1 -8370,E2 -8370} C_VEL
LIN {X 0,Y 452.562,Z 860.49,A -85,B 0,C 180,E1 -8370.889,E2 -8370.889} C_VEL
LIN {X 0,Y 452.575,Z 858.837,A -85,B 0,C 180,E1 -8372.67,E2 -8372.67} C_VEL
LIN {X 0,Y 452.58,Z 857.384,A -85,B 0,C 180,E1 -8373.561,E2 -8373.561} C_VEL
LIN {X 0,Y 452.626,Z 854.366,A -85,B 0,C 180,E1 -8374.898,E2 -8374.898} C_VEL
LIN {X 0,Y 452.691,Z 849.368,A -85,B 0,C 180,E1 -8376.485,E2 -8376.485} C_VEL
LIN {X 0,Y 452.907,Z 842.928,A -85,B 0,C 180,E1 -8378.027,E2 -8378.027} C_VEL
LIN {X 0,Y 453.197,Z 835.736,A -85,B 0,C 180,E1 -8379.371,E2 -8379.371} C_VEL
LIN {X 0,Y 453.526,Z 826.772,A -85,B 0,C 180,E1 -8380.716,E2 -8380.716} C_VEL
LIN {X 0,Y 454.029,Z 817.538,A -85,B 0,C 180,E1 -8381.835,E2 -8381.835} C_VEL
LIN {X 0,Y 454.552,Z 806.57,A -85,B 0,C 180,E1 -8382.898,E2 -8382.898} C_VEL
LIN {X 0,Y 455.014,Z 795.772,A -85,B 0,C 180,E1 -8383.737,E2 -8383.737} C_VEL
LIN {X 0,Y 455.538,Z 783.739,A -85,B 0,C 180,E1 -8384.461,E2 -8384.461} C_VEL
LIN {X 0,Y 455.944,Z 771.308,A -85,B 0,C 180,E1 -8385.076,E2 -8385.076} C_VEL
LIN {X 0,Y 454.576,Z 759.255,A -85,B 0,C 180,E1 -8385.567,E2 -8385.567} C_VEL
LIN {X 0,Y 453.298,Z 746.128,A -85,B 0,C 180,E1 -8385.939,E2 -8385.939} C_VEL
LIN {X 0,Y 453.633,Z 732.519,A -85,B 0,C 180,E1 -8389.081,E2 -8389.081} C_VEL
LIN {X 0,Y 454.035,Z 718.818,A -85,B 0,C 180,E1 -8392.286,E2 -8392.286} C_VEL
LIN {X 0,Y 454.523,Z 705.689,A -85,B 0,C 180,E1 -8395.408,E2 -8395.408} C_VEL
LIN {X 0,Y 455.146,Z 691.556,A -85,B 0,C 180,E1 -8398.85,E2 -8398.85} C_VEL
LIN {X 0,Y 455.81,Z 677.887,A -85,B 0,C 180,E1 -8402.273,E2 -8402.273} C_VEL
LIN {X 0,Y 456.415,Z 667.219,A -85,B 0,C 180,E1 -8405.023,E2 -8405.023} C_VEL
LIN {X 0,Y 456.668,Z 660.24,A -85,B 0,C 180,E1 -8406.883,E2 -8406.883} C_VEL
LIN {X 0,Y 455.004,Z 651.414,A -85,B 0,C 180,E1 -8409.439,E2 -8409.439} C_VEL
LIN {X 0,Y 453.486,Z 643.998,A -85,B 0,C 180,E1 -8411.71,E2 -8411.71} C_VEL
LIN {X 0,Y 453.485,Z 643.999,A -85,B 0,C 180,E1 -8414.529,E2 -8414.529} C_VEL
LIN {X 0,Y 453.494,Z 643.997,A -85,B 0,C 180,E1 -8418.062,E2 -8418.062} C_VEL
LIN {X 0,Y 453.53,Z 643.992,A -85,B 0,C 180,E1 -8420.787,E2 -8420.787} C_VEL
LIN {X 0,Y 453.453,Z 644.002,A -85,B 0,C 180,E1 -8423.917,E2 -8423.917} C_VEL
LIN {X 0,Y 453.479,Z 643.996,A -85,B 0,C 180,E1 -8427.151,E2 -8427.151} C_VEL
LIN {X 0,Y 453.51,Z 643.992,A -85,B 0,C 180,E1 -8430.271,E2 -8430.271} C_VEL
LIN {X 0,Y 453.51,Z 643.995,A -85,B 0,C 180,E1 -8433.294,E2 -8433.294} C_VEL
LIN {X 0,Y 453.499,Z 643.993,A -85,B 0,C 180,E1 -8436.238,E2 -8436.238} C_VEL
LIN {X 0,Y 453.479,Z 644,A -85,B 0,C 180,E1 -8439.117,E2 -8439.117} C_VEL
LIN {X 0,Y 453.506,Z 643.991,A -85,B 0,C 180,E1 -8441.944,E2 -8441.944} C_VEL
LIN {X 0,Y 453.535,Z 643.991,A -85,B 0,C 180,E1 -8444.726,E2 -8444.726} C_VEL
LIN {X 0,Y 453.597,Z 643.983,A -85,B 0,C 180,E1 -8447.472,E2 -8447.472} C_VEL
LIN {X 0,Y 453.589,Z 643.985,A -85,B 0,C 180,E1 -8451.086,E2 -8451.086} C_VEL
LIN {X 0,Y 453.672,Z 643.974,A -85,B 0,C 180,E1 -8453.774,E2 -8453.774} C_VEL
LIN {X 0,Y 453.76,Z 643.962,A -85,B 0,C 180,E1 -8457.337,E2 -8457.337} C_VEL
LIN {X 0,Y 453.818,Z 643.96,A -85,B 0,C 180,E1 -8460,E2 -8460} C_VEL
LIN {X 0,Y 453.783,Z 644.007,A -85,B 0,C 180,E1 -8462.607,E2 -8462.607} C_VEL
LIN {X 0,Y 454.917,Z 652.515,A -85,B 0,C 180,E1 -8464.874,E2 -8464.874} C_VEL
LIN {X 0,Y 455.019,Z 662.719,A -85,B 0,C 180,E1 -8467.544,E2 -8467.544} C_VEL
LIN {X 0,Y 454.792,Z 672.872,A -85,B 0,C 180,E1 -8470.236,E2 -8470.236} C_VEL
LIN {X 0,Y 454.67,Z 683.667,A -85,B 0,C 180,E1 -8473.145,E2 -8473.145} C_VEL
LIN {X 0,Y 454.34,Z 694.666,A -85,B 0,C 180,E1 -8476.167,E2 -8476.167} C_VEL
LIN {X 0,Y 454.108,Z 704.995,A -85,B 0,C 180,E1 -8478.966,E2 -8478.966} C_VEL
LIN {X 0,Y 453.788,Z 717.002,A -85,B 0,C 180,E1 -8482.299,E2 -8482.299} C_VEL
LIN {X 0,Y 453.549,Z 727.371,A -85,B 0,C 180,E1 -8485.161,E2 -8485.161} C_VEL
LIN {X 0,Y 455.993,Z 740.656,A -85,B 0,C 180,E1 -8485.592,E2 -8485.592} C_VEL
LIN {X 0,Y 456.527,Z 745.887,A -85,B 0,C 180,E1 -8485.8,E2 -8485.8} C_VEL
LIN {X 0,Y 456.107,Z 758.199,A -85,B 0,C 180,E1 -8486.359,E2 -8486.359} C_VEL
LIN {X 0,Y 455.541,Z 770.3,A -85,B 0,C 180,E1 -8487.091,E2 -8487.091} C_VEL
LIN {X 0,Y 454.982,Z 782.175,A -85,B 0,C 180,E1 -8488.034,E2 -8488.034} C_VEL
LIN {X 0,Y 454.422,Z 792.198,A -85,B 0,C 180,E1 -8489.028,E2 -8489.028} C_VEL
LIN {X 0,Y 453.879,Z 802.057,A -85,B 0,C 180,E1 -8490.24,E2 -8490.24} C_VEL
LIN {X 0,Y 453.447,Z 810.43,A -85,B 0,C 180,E1 -8491.523,E2 -8491.523} C_VEL
LIN {X 0,Y 453.08,Z 817.614,A -85,B 0,C 180,E1 -8492.882,E2 -8492.882} C_VEL
LIN {X 0,Y 452.803,Z 823.551,A -85,B 0,C 180,E1 -8494.3,E2 -8494.3} C_VEL
LIN {X 0,Y 452.628,Z 827.808,A -85,B 0,C 180,E1 -8495.602,E2 -8495.602} C_VEL
LIN {X 0,Y 452.473,Z 831.797,A -85,B 0,C 180,E1 -8497.284,E2 -8497.284} C_VEL
LIN {X 0,Y 452.333,Z 834.355,A -85,B 0,C 180,E1 -8499.027,E2 -8499.027} C_VEL
LIN {X 0,Y 452.286,Z 835.326,A -85,B 0,C 180,E1 -8500.74,E2 -8500.74} C_VEL
LIN {X 0,Y 452.281,Z 835.154,A -85,B 0,C 180,E1 -8501.927,E2 -8501.927} C_VEL
LIN {X 0,Y 452.321,Z 834.266,A -85,B 0,C 180,E1 -8503.13,E2 -8503.13} C_VEL
LIN {X 0,Y 452.437,Z 831.421,A -85,B 0,C 180,E1 -8504.973,E2 -8504.973} C_VEL
LIN {X 0,Y 452.579,Z 828.275,A -85,B 0,C 180,E1 -8506.29,E2 -8506.29} C_VEL
LIN {X 0,Y 452.816,Z 823.29,A -85,B 0,C 180,E1 -8507.836,E2 -8507.836} C_VEL
LIN {X 0,Y 453.081,Z 816.825,A -85,B 0,C 180,E1 -8509.347,E2 -8509.347} C_VEL
LIN {X 0,Y 453.49,Z 808.957,A -85,B 0,C 180,E1 -8510.794,E2 -8510.794} C_VEL
LIN {X 0,Y 453.88,Z 801.063,A -85,B 0,C 180,E1 -8511.965,E2 -8511.965} C_VEL
LIN {X 0,Y 454.417,Z 791.971,A -85,B 0,C 180,E1 -8513.065,E2 -8513.065} C_VEL
LIN {X 0,Y 454.985,Z 780.758,A -85,B 0,C 180,E1 -8514.165,E2 -8514.165} C_VEL
LIN {X 0,Y 455.547,Z 769.44,A -85,B 0,C 180,E1 -8515.04,E2 -8515.04} C_VEL
LIN {X 0,Y 456.127,Z 757.368,A -85,B 0,C 180,E1 -8515.76,E2 -8515.76} C_VEL
LIN {X 0,Y 456.48,Z 744.274,A -85,B 0,C 180,E1 -8516.341,E2 -8516.341} C_VEL
LIN {X 0,Y 454.28,Z 731.23,A -85,B 0,C 180,E1 -8516.807,E2 -8516.807} C_VEL
LIN {X 0,Y 453.489,Z 726.935,A -85,B 0,C 180,E1 -8516.941,E2 -8516.941} C_VEL
LIN {X 0,Y 453.825,Z 715.086,A -85,B 0,C 180,E1 -8520.294,E2 -8520.294} C_VEL
LIN {X 0,Y 454.111,Z 706.083,A -85,B 0,C 180,E1 -8522.836,E2 -8522.836} C_VEL
LIN {X 0,Y 454.438,Z 695.426,A -85,B 0,C 180,E1 -8525.846,E2 -8525.846} C_VEL
LIN {X 0,Y 454.485,Z 693.766,A -85,B 0,C 180,E1 -8526.318,E2 -8526.318} C_VEL
LIN {X 0,Y 453.892,Z 691.479,A -85,B 0,C 180,E1 -8527,E2 -8527} C_VEL
LIN {X 0,Y 451.189,Z 688.037,A -85,B 0,C 180,E1 -8528.126,E2 -8528.126} C_VEL
LIN {X 0,Y 448.906,Z 685.296,A -85,B 0,C 180,E1 -8529.035,E2 -8529.035} C_VEL
LIN {X 0,Y 447.963,Z 683.059,A -85,B 0,C 180,E1 -8529.729,E2 -8529.729} C_VEL
LIN {X 0,Y 447.906,Z 682.26,A -85,B 0,C 180,E1 -8529.961,E2 -8529.961} C_VEL
LIN {X 0,Y 448.187,Z 671.452,A -85,B 0,C 180,E1 -8533.046,E2 -8533.046} C_VEL
LIN {X 0,Y 448.414,Z 661.109,A -85,B 0,C 180,E1 -8535.987,E2 -8535.987} C_VEL
LIN {X 0,Y 448.241,Z 654.885,A -85,B 0,C 180,E1 -8537.781,E2 -8537.781} C_VEL
LIN {X 0,Y 446.991,Z 647.303,A -85,B 0,C 180,E1 -8540.041,E2 -8540.041} C_VEL
LIN {X 0,Y 446.562,Z 644.862,A -85,B 0,C 180,E1 -8540.832,E2 -8540.832} C_VEL
LIN {X 0,Y 446.646,Z 644.853,A -85,B 0,C 180,E1 -8543.677,E2 -8543.677} C_VEL
LIN {X 0,Y 446.711,Z 644.844,A -85,B 0,C 180,E1 -8547.295,E2 -8547.295} C_VEL
LIN {X 0,Y 446.796,Z 644.832,A -85,B 0,C 180,E1 -8550,E2 -8550} C_VEL
LIN {X 0,Y 446.711,Z 644.842,A -85,B 0,C 180,E1 -8552.706,E2 -8552.706} C_VEL
LIN {X 0,Y 446.64,Z 644.848,A -85,B 0,C 180,E1 -8556.324,E2 -8556.324} C_VEL
LIN {X 0,Y 446.541,Z 644.861,A -85,B 0,C 180,E1 -8559.056,E2 -8559.056} C_VEL
LIN {X 0,Y 446.536,Z 644.865,A -85,B 0,C 180,E1 -8562.73,E2 -8562.73} C_VEL
LIN {X 0,Y 446.492,Z 644.871,A -85,B 0,C 180,E1 -8566.459,E2 -8566.459} C_VEL
LIN {X 0,Y 446.471,Z 644.875,A -85,B 0,C 180,E1 -8569.303,E2 -8569.303} C_VEL
LIN {X 0,Y 446.456,Z 644.877,A -85,B 0,C 180,E1 -8572.747,E2 -8572.747} C_VEL
LIN {X 0,Y 449.675,Z 656.042,A -85,B 0,C 180,E1 -8573.487,E2 -8573.487} C_VEL
LIN {X 0,Y 449.698,Z 661.493,A -85,B 0,C 180,E1 -8573.853,E2 -8573.853} C_VEL
LIN {X 0,Y 449.267,Z 672.534,A -85,B 0,C 180,E1 -8574.72,E2 -8574.72} C_VEL
LIN {X 0,Y 448.764,Z 683.141,A -85,B 0,C 180,E1 -8575.759,E2 -8575.759} C_VEL
LIN {X 0,Y 448.308,Z 691.899,A -85,B 0,C 180,E1 -8576.814,E2 -8576.814} C_VEL
LIN {X 0,Y 447.818,Z 700.522,A -85,B 0,C 180,E1 -8578.088,E2 -8578.088} C_VEL
LIN {X 0,Y 447.356,Z 707.718,A -85,B 0,C 180,E1 -8579.399,E2 -8579.399} C_VEL
LIN {X 0,Y 446.944,Z 714.672,A -85,B 0,C 180,E1 -8580.996,E2 -8580.996} C_VEL
LIN {X 0,Y 446.738,Z 719.163,A -85,B 0,C 180,E1 -8582.336,E2 -8582.336} C_VEL
LIN {X 0,Y 446.48,Z 723.226,A -85,B 0,C 180,E1 -8583.973,E2 -8583.973} C_VEL
LIN {X 0,Y 446.264,Z 725.952,A -85,B 0,C 180,E1 -8585.641,E2 -8585.641} C_VEL
LIN {X 0,Y 446.231,Z 727.008,A -85,B 0,C 180,E1 -8586.762,E2 -8586.762} C_VEL
LIN {X 0,Y 446.236,Z 727.493,A -85,B 0,C 180,E1 -8588.05,E2 -8588.05} C_VEL
LIN {X 0,Y 446.306,Z 727.071,A -85,B 0,C 180,E1 -8589.502,E2 -8589.502} C_VEL
LIN {X 0,Y 446.377,Z 725.705,A -85,B 0,C 180,E1 -8590.91,E2 -8590.91} C_VEL
LIN {X 0,Y 446.596,Z 722.763,A -85,B 0,C 180,E1 -8592.585,E2 -8592.585} C_VEL
LIN {X 0,Y 446.809,Z 719.743,A -85,B 0,C 180,E1 -8593.796,E2 -8593.796} C_VEL
LIN {X 0,Y 447.121,Z 714.619,A -85,B 0,C 180,E1 -8595.337,E2 -8595.337} C_VEL
LIN {X 0,Y 447.597,Z 707.849,A -85,B 0,C 180,E1 -8596.896,E2 -8596.896} C_VEL
LIN {X 0,Y 448.066,Z 700.698,A -85,B 0,C 180,E1 -8598.194,E2 -8598.194} C_VEL
LIN {X 0,Y 448.551,Z 692.199,A -85,B 0,C 180,E1 -8599.441,E2 -8599.441} C_VEL
LIN {X 0,Y 449.121,Z 682.994,A -85,B 0,C 180,E1 -8600.537,E2 -8600.537} C_VEL
LIN {X 0,Y 449.584,Z 672.809,A -85,B 0,C 180,E1 -8601.527,E2 -8601.527} C_VEL
LIN {X 0,Y 450.011,Z 661.342,A -85,B 0,C 180,E1 -8602.407,E2 -8602.407} C_VEL
LIN {X 0,Y 450.165,Z 657.654,A -85,B 0,C 180,E1 -8602.647,E2 -8602.647} C_VEL
LIN {X 0,Y 447.286,Z 647.615,A -85,B 0,C 180,E1 -8603.339,E2 -8603.339} C_VEL
LIN {X 0,Y 446.424,Z 644.877,A -85,B 0,C 180,E1 -8603.522,E2 -8603.522} C_VEL
LIN {X 0,Y 446.449,Z 644.872,A -85,B 0,C 180,E1 -8606.567,E2 -8606.567} C_VEL
LIN {X 0,Y 446.431,Z 644.876,A -85,B 0,C 180,E1 -8609.979,E2 -8609.979} C_VEL
LIN {X 0,Y 446.473,Z 644.868,A -85,B 0,C 180,E1 -8612.839,E2 -8612.839} C_VEL
LIN {X 0,Y 446.463,Z 644.87,A -85,B 0,C 180,E1 -8615.925,E2 -8615.925} C_VEL
LIN {X 0,Y 446.454,Z 644.871,A -85,B 0,C 180,E1 -8618.773,E2 -8618.773} C_VEL
LIN {X 0,Y 446.459,Z 644.876,A -85,B 0,C 180,E1 -8621.649,E2 -8621.649} C_VEL
LIN {X 0,Y 446.517,Z 644.864,A -85,B 0,C 180,E1 -8624.48,E2 -8624.48} C_VEL
LIN {X 0,Y 446.519,Z 644.862,A -85,B 0,C 180,E1 -8628.193,E2 -8628.193} C_VEL
LIN {X 0,Y 446.602,Z 644.853,A -85,B 0,C 180,E1 -8631.858,E2 -8631.858} C_VEL
LIN {X 0,Y 446.647,Z 644.846,A -85,B 0,C 180,E1 -8634.583,E2 -8634.583} C_VEL
LIN {X 0,Y 446.71,Z 644.833,A -85,B 0,C 180,E1 -8637.295,E2 -8637.295} C_VEL
LIN {X 0,Y 446.795,Z 644.829,A -85,B 0,C 180,E1 -8640,E2 -8640} C_VEL
LIN {X 0,Y 446.711,Z 644.838,A -85,B 0,C 180,E1 -8642.705,E2 -8642.705} C_VEL
LIN {X 0,Y 446.648,Z 644.851,A -85,B 0,C 180,E1 -8646.324,E2 -8646.324} C_VEL
LIN {X 0,Y 446.54,Z 644.854,A -85,B 0,C 180,E1 -8649.055,E2 -8649.055} C_VEL
LIN {X 0,Y 446.523,Z 644.859,A -85,B 0,C 180,E1 -8652.73,E2 -8652.73} C_VEL
LIN {X 0,Y 446.498,Z 644.867,A -85,B 0,C 180,E1 -8656.228,E2 -8656.228} C_VEL
LIN {X 0,Y 446.471,Z 644.865,A -85,B 0,C 180,E1 -8659.303,E2 -8659.303} C_VEL
LIN {X 0,Y 446.42,Z 644.879,A -85,B 0,C 180,E1 -8662.2,E2 -8662.2} C_VEL
LIN {X 0,Y 446.459,Z 644.868,A -85,B 0,C 180,E1 -8665.152,E2 -8665.152} C_VEL
LIN {X 0,Y 446.487,Z 644.87,A -85,B 0,C 180,E1 -8668.179,E2 -8668.179} C_VEL
LIN {X 0,Y 446.421,Z 644.875,A -85,B 0,C 180,E1 -8671.775,E2 -8671.775} C_VEL
LIN {X 0,Y 446.431,Z 644.878,A -85,B 0,C 180,E1 -8674.523,E2 -8674.523} C_VEL
LIN {X 0,Y 446.418,Z 644.879,A -85,B 0,C 180,E1 -8678.079,E2 -8678.079} C_VEL
LIN {X 0,Y 446.429,Z 644.878,A -85,B 0,C 180,E1 -8680.918,E2 -8680.918} C_VEL
LIN {X 0,Y 446.404,Z 644.877,A -85,B 0,C 180,E1 -8683.846,E2 -8683.846} C_VEL
LIN {X 0,Y 446.402,Z 644.884,A -85,B 0,C 180,E1 -8686.403,E2 -8686.403} C_VEL
LIN {X 0,Y 446.477,Z 645.058,A -85,B 0,C 180,E1 -8688.614,E2 -8688.614} C_VEL
LIN {X 0,Y 448.379,Z 654.582,A -85,B 0,C 180,E1 -8691.602,E2 -8691.602} C_VEL
LIN {X 0,Y 449.297,Z 660.131,A -85,B 0,C 180,E1 -8693.24,E2 -8693.24} C_VEL
LIN {X 0,Y 448.902,Z 668.179,A -85,B 0,C 180,E1 -8695.422,E2 -8695.422} C_VEL
LIN {X 0,Y 448.286,Z 680.305,A -85,B 0,C 180,E1 -8698.583,E2 -8698.583} C_VEL
LIN {X 0,Y 447.706,Z 693.537,A -85,B 0,C 180,E1 -8701.905,E2 -8701.905} C_VEL
LIN {X 0,Y 447.25,Z 705.863,A -85,B 0,C 180,E1 -8704.895,E2 -8704.895} C_VEL
LIN {X 0,Y 446.811,Z 718.129,A -85,B 0,C 180,E1 -8707.821,E2 -8707.821} C_VEL
LIN {X 0,Y 446.489,Z 732.703,A -85,B 0,C 180,E1 -8711.228,E2 -8711.228} C_VEL
LIN {X 0,Y 446.239,Z 743.834,A -85,B 0,C 180,E1 -8713.8,E2 -8713.8} C_VEL
LIN {X 0,Y 447.546,Z 758.353,A -85,B 0,C 180,E1 -8714.216,E2 -8714.216} C_VEL
LIN {X 0,Y 448.948,Z 773.95,A -85,B 0,C 180,E1 -8714.856,E2 -8714.856} C_VEL
LIN {X 0,Y 448.554,Z 786.687,A -85,B 0,C 180,E1 -8715.481,E2 -8715.481} C_VEL
LIN {X 0,Y 447.946,Z 798.837,A -85,B 0,C 180,E1 -8716.272,E2 -8716.272} C_VEL
LIN {X 0,Y 447.501,Z 809.005,A -85,B 0,C 180,E1 -8717.12,E2 -8717.12} C_VEL
LIN {X 0,Y 446.981,Z 819.429,A -85,B 0,C 180,E1 -8718.205,E2 -8718.205} C_VEL
LIN {X 0,Y 446.484,Z 828.325,A -85,B 0,C 180,E1 -8719.341,E2 -8719.341} C_VEL
LIN {X 0,Y 446.144,Z 835.651,A -85,B 0,C 180,E1 -8720.479,E2 -8720.479} C_VEL
LIN {X 0,Y 445.875,Z 842.831,A -85,B 0,C 180,E1 -8721.844,E2 -8721.844} C_VEL
LIN {X 0,Y 445.646,Z 849.505,A -85,B 0,C 180,E1 -8723.483,E2 -8723.483} C_VEL
LIN {X 0,Y 445.565,Z 854.227,A -85,B 0,C 180,E1 -8725.023,E2 -8725.023} C_VEL
LIN {X 0,Y 445.484,Z 857.229,A -85,B 0,C 180,E1 -8726.382,E2 -8726.382} C_VEL
LIN {X 0,Y 445.499,Z 858.673,A -85,B 0,C 180,E1 -8727.287,E2 -8727.287} C_VEL
LIN {X 0,Y 445.469,Z 860.301,A -85,B 0,C 180,E1 -8729.096,E2 -8729.096} C_VEL
LIN {X 0,Y 445.476,Z 860.52,A -85,B 0,C 180,E1 -8730,E2 -8730} C_VEL
LIN {X 0,Y 445.465,Z 860.29,A -85,B 0,C 180,E1 -8730.903,E2 -8730.903} C_VEL
LIN {X 0,Y 445.498,Z 858.636,A -85,B 0,C 180,E1 -8732.712,E2 -8732.712} C_VEL
LIN {X 0,Y 445.477,Z 857.181,A -85,B 0,C 180,E1 -8733.618,E2 -8733.618} C_VEL
LIN {X 0,Y 445.553,Z 854.162,A -85,B 0,C 180,E1 -8734.976,E2 -8734.976} C_VEL
LIN {X 0,Y 445.605,Z 849.584,A -85,B 0,C 180,E1 -8736.471,E2 -8736.471} C_VEL
LIN {X 0,Y 445.796,Z 843.739,A -85,B 0,C 180,E1 -8737.928,E2 -8737.928} C_VEL
LIN {X 0,Y 446.088,Z 836.842,A -85,B 0,C 180,E1 -8739.293,E2 -8739.293} C_VEL
LIN {X 0,Y 446.407,Z 829.79,A -85,B 0,C 180,E1 -8740.43,E2 -8740.43} C_VEL
LIN {X 0,Y 446.899,Z 821.254,A -85,B 0,C 180,E1 -8741.566,E2 -8741.566} C_VEL
LIN {X 0,Y 447.414,Z 810.68,A -85,B 0,C 180,E1 -8742.703,E2 -8742.703} C_VEL
LIN {X 0,Y 447.857,Z 800.191,A -85,B 0,C 180,E1 -8743.614,E2 -8743.614} C_VEL
LIN {X 0,Y 448.43,Z 788.575,A -85,B 0,C 180,E1 -8744.406,E2 -8744.406} C_VEL
LIN {X 0,Y 448.896,Z 775.247,A -85,B 0,C 180,E1 -8745.086,E2 -8745.086} C_VEL
LIN {X 0,Y 448.925,Z 771.564,A -85,B 0,C 180,E1 -8745.26,E2 -8745.26} C_VEL
LIN {X 0,Y 447.61,Z 759.155,A -85,B 0,C 180,E1 -8745.783,E2 -8745.783} C_VEL
LIN {X 0,Y 446.242,Z 745.257,A -85,B 0,C 180,E1 -8746.183,E2 -8746.183} C_VEL
LIN {X 0,Y 446.589,Z 731.012,A -85,B 0,C 180,E1 -8749.536,E2 -8749.536} C_VEL
LIN {X 0,Y 447.037,Z 716.937,A -85,B 0,C 180,E1 -8752.898,E2 -8752.898} C_VEL
LIN {X 0,Y 447.547,Z 704.868,A -85,B 0,C 180,E1 -8755.833,E2 -8755.833} C_VEL
LIN {X 0,Y 448.188,Z 690.746,A -85,B 0,C 180,E1 -8759.342,E2 -8759.342} C_VEL
LIN {X 0,Y 448.797,Z 679.316,A -85,B 0,C 180,E1 -8762.261,E2 -8762.261} C_VEL
LIN {X 0,Y 449.5,Z 667.571,A -85,B 0,C 180,E1 -8765.344,E2 -8765.344} C_VEL
LIN {X 0,Y 449.772,Z 662.279,A -85,B 0,C 180,E1 -8766.776,E2 -8766.776} C_VEL
LIN {X 0,Y 448.238,Z 653.73,A -85,B 0,C 180,E1 -8769.278,E2 -8769.278} C_VEL
LIN {X 0,Y 446.421,Z 644.879,A -85,B 0,C 180,E1 -8772.042,E2 -8772.042} C_VEL
LIN {X 0,Y 446.454,Z 644.874,A -85,B 0,C 180,E1 -8775.102,E2 -8775.102} C_VEL
LIN {X 0,Y 446.441,Z 644.877,A -85,B 0,C 180,E1 -8778.61,E2 -8778.61} C_VEL
LIN {X 0,Y 446.473,Z 644.869,A -85,B 0,C 180,E1 -8780.976,E2 -8780.976} C_VEL
LIN {X 0,Y 446.417,Z 644.877,A -85,B 0,C 180,E1 -8784.374,E2 -8784.374} C_VEL
LIN {X 0,Y 446.419,Z 644.878,A -85,B 0,C 180,E1 -8787.638,E2 -8787.638} C_VEL
LIN {X 0,Y 446.465,Z 644.867,A -85,B 0,C 180,E1 -8790.792,E2 -8790.792} C_VEL
LIN {X 0,Y 446.473,Z 644.868,A -85,B 0,C 180,E1 -8793.848,E2 -8793.848} C_VEL
LIN {X 0,Y 446.425,Z 644.874,A -85,B 0,C 180,E1 -8796.823,E2 -8796.823} C_VEL
LIN {X 0,Y 446.44,Z 644.872,A -85,B 0,C 180,E1 -8799.737,E2 -8799.737} C_VEL
LIN {X 0,Y 446.458,Z 644.869,A -85,B 0,C 180,E1 -8802.597,E2 -8802.597} C_VEL
LIN {X 0,Y 446.467,Z 644.873,A -85,B 0,C 180,E1 -8805.412,E2 -8805.412} C_VEL
LIN {X 0,Y 446.541,Z 644.861,A -85,B 0,C 180,E1 -8808.194,E2 -8808.194} C_VEL
LIN {X 0,Y 446.595,Z 644.855,A -85,B 0,C 180,E1 -8811.858,E2 -8811.858} C_VEL
LIN {X 0,Y 446.64,Z 644.852,A -85,B 0,C 180,E1 -8814.582,E2 -8814.582} C_VEL
LIN {X 0,Y 446.704,Z 644.842,A -85,B 0,C 180,E1 -8817.295,E2 -8817.295} C_VEL
LIN {X 0,Y 446.788,Z 644.836,A -85,B 0,C 180,E1 -8820,E2 -8820} C_VEL
LIN {X 0,Y 446.725,Z 645.035,A -85,B 0,C 180,E1 -8822.367,E2 -8822.367} C_VEL
LIN {X 0,Y 448.054,Z 654.583,A -85,B 0,C 180,E1 -8824.949,E2 -8824.949} C_VEL
LIN {X 0,Y 448.085,Z 664.803,A -85,B 0,C 180,E1 -8827.661,E2 -8827.661} C_VEL
LIN {X 0,Y 447.833,Z 675.068,A -85,B 0,C 180,E1 -8830.397,E2 -8830.397} C_VEL
LIN {X 0,Y 447.657,Z 685.533,A -85,B 0,C 180,E1 -8833.256,E2 -8833.256} C_VEL
LIN {X 0,Y 447.383,Z 695.344,A -85,B 0,C 180,E1 -8835.957,E2 -8835.957} C_VEL
LIN {X 0,Y 447.131,Z 705.667,A -85,B 0,C 180,E1 -8838.797,E2 -8838.797} C_VEL
LIN {X 0,Y 446.815,Z 716.664,A -85,B 0,C 180,E1 -8841.875,E2 -8841.875} C_VEL
LIN {X 0,Y 446.545,Z 727.496,A -85,B 0,C 180,E1 -8844.898,E2 -8844.898} C_VEL
LIN {X 0,Y 449.024,Z 740.672,A -85,B 0,C 180,E1 -8845.339,E2 -8845.339} C_VEL
LIN {X 0,Y 449.684,Z 746.455,A -85,B 0,C 180,E1 -8845.578,E2 -8845.578} C_VEL
LIN {X 0,Y 449.224,Z 758.961,A -85,B 0,C 180,E1 -8846.162,E2 -8846.162} C_VEL
LIN {X 0,Y 448.619,Z 771.431,A -85,B 0,C 180,E1 -8846.942,E2 -8846.942} C_VEL
LIN {X 0,Y 448.068,Z 782.199,A -85,B 0,C 180,E1 -8847.816,E2 -8847.816} C_VEL
LIN {X 0,Y 447.521,Z 791.659,A -85,B 0,C 180,E1 -8848.76,E2 -8848.76} C_VEL
LIN {X 0,Y 446.961,Z 801.025,A -85,B 0,C 180,E1 -8849.901,E2 -8849.901} C_VEL
LIN {X 0,Y 446.538,Z 808.606,A -85,B 0,C 180,E1 -8851.027,E2 -8851.027} C_VEL
LIN {X 0,Y 446.144,Z 816.043,A -85,B 0,C 180,E1 -8852.384,E2 -8852.384} C_VEL
LIN {X 0,Y 445.857,Z 822.076,A -85,B 0,C 180,E1 -8853.755,E2 -8853.755} C_VEL
LIN {X 0,Y 445.573,Z 827.296,A -85,B 0,C 180,E1 -8855.271,E2 -8855.271} C_VEL
LIN {X 0,Y 445.414,Z 831.261,A -85,B 0,C 180,E1 -8856.84,E2 -8856.84} C_VEL
LIN {X 0,Y 445.333,Z 833.293,A -85,B 0,C 180,E1 -8857.986,E2 -8857.986} C_VEL
LIN {X 0,Y 445.236,Z 834.851,A -85,B 0,C 180,E1 -8859.336,E2 -8859.336} C_VEL
LIN {X 0,Y 445.206,Z 835.526,A -85,B 0,C 180,E1 -8860.737,E2 -8860.737} C_VEL
LIN {X 0,Y 445.18,Z 835.266,A -85,B 0,C 180,E1 -8862.101,E2 -8862.101} C_VEL
LIN {X 0,Y 445.276,Z 833.428,A -85,B 0,C 180,E1 -8863.985,E2 -8863.985} C_VEL
LIN {X 0,Y 445.377,Z 831.202,A -85,B 0,C 180,E1 -8865.243,E2 -8865.243} C_VEL
LIN {X 0,Y 445.584,Z 826.89,A -85,B 0,C 180,E1 -8866.916,E2 -8866.916} C_VEL
LIN {X 0,Y 445.817,Z 821.14,A -85,B 0,C 180,E1 -8868.541,E2 -8868.541} C_VEL
LIN {X 0,Y 446.152,Z 814.59,A -85,B 0,C 180,E1 -8869.964,E2 -8869.964} C_VEL
LIN {X 0,Y 446.552,Z 807.433,A -85,B 0,C 180,E1 -8871.216,E2 -8871.216} C_VEL
LIN {X 0,Y 447.083,Z 798.699,A -85,B 0,C 180,E1 -8872.462,E2 -8872.462} C_VEL
LIN {X 0,Y 447.693,Z 788.312,A -85,B 0,C 180,E1 -8873.659,E2 -8873.659} C_VEL
LIN {X 0,Y 448.298,Z 776.992,A -85,B 0,C 180,E1 -8874.695,E2 -8874.695} C_VEL
LIN {X 0,Y 448.863,Z 766.081,A -85,B 0,C 180,E1 -8875.487,E2 -8875.487} C_VEL
LIN {X 0,Y 449.434,Z 753.214,A -85,B 0,C 180,E1 -8876.198,E2 -8876.198} C_VEL
LIN {X 0,Y 449.53,Z 744.536,A -85,B 0,C 180,E1 -8876.573,E2 -8876.573} C_VEL
LIN {X 0,Y 447.356,Z 731.558,A -85,B 0,C 180,E1 -8877.047,E2 -8877.047} C_VEL
LIN {X 0,Y 446.489,Z 727.079,A -85,B 0,C 180,E1 -8877.193,E2 -8877.193} C_VEL
LIN {X 0,Y 446.885,Z 714.332,A -85,B 0,C 180,E1 -8880.823,E2 -8880.823} C_VEL
LIN {X 0,Y 447.204,Z 703.546,A -85,B 0,C 180,E1 -8883.895,E2 -8883.895} C_VEL
LIN {X 0,Y 447.562,Z 693.046,A -85,B 0,C 180,E1 -8886.886,E2 -8886.886} C_VEL
LIN {X 0,Y 447.906,Z 682.26,A -85,B 0,C 180,E1 -8889.961,E2 -8889.961} C_VEL
LIN {X 0,Y 447.31,Z 679.968,A -85,B 0,C 180,E1 -8890.653,E2 -8890.653} C_VEL
LIN {X 0,Y 444.569,Z 676.568,A -85,B 0,C 180,E1 -8891.798,E2 -8891.798} C_VEL
LIN {X 0,Y 442.263,Z 673.866,A -85,B 0,C 180,E1 -8892.722,E2 -8892.722} C_VEL
LIN {X 0,Y 441.323,Z 671.633,A -85,B 0,C 180,E1 -8893.425,E2 -8893.425} C_VEL
LIN {X 0,Y 441.274,Z 670.822,A -85,B 0,C 180,E1 -8893.66,E2 -8893.66} C_VEL
LIN {X 0,Y 441.503,Z 660.394,A -85,B 0,C 180,E1 -8896.655,E2 -8896.655} C_VEL
LIN {X 0,Y 441.024,Z 654.093,A -85,B 0,C 180,E1 -8898.511,E2 -8898.511} C_VEL
LIN {X 0,Y 439.5,Z 645.741,A -85,B 0,C 180,E1 -8901.089,E2 -8901.089} C_VEL
LIN {X 0,Y 439.619,Z 645.728,A -85,B 0,C 180,E1 -8903.575,E2 -8903.575} C_VEL
LIN {X 0,Y 439.658,Z 645.723,A -85,B 0,C 180,E1 -8907.252,E2 -8907.252} C_VEL
LIN {X 0,Y 439.766,Z 645.708,A -85,B 0,C 180,E1 -8910,E2 -8910} C_VEL
LIN {X 0,Y 439.658,Z 645.72,A -85,B 0,C 180,E1 -8912.749,E2 -8912.749} C_VEL
LIN {X 0,Y 439.615,Z 645.723,A -85,B 0,C 180,E1 -8916.426,E2 -8916.426} C_VEL
LIN {X 0,Y 439.503,Z 645.737,A -85,B 0,C 180,E1 -8919.202,E2 -8919.202} C_VEL
LIN {X 0,Y 439.506,Z 645.741,A -85,B 0,C 180,E1 -8922.727,E2 -8922.727} C_VEL
LIN {X 0,Y 439.449,Z 645.747,A -85,B 0,C 180,E1 -8926.349,E2 -8926.349} C_VEL
LIN {X 0,Y 439.404,Z 645.755,A -85,B 0,C 180,E1 -8929.627,E2 -8929.627} C_VEL
LIN {X 0,Y 439.399,Z 645.754,A -85,B 0,C 180,E1 -8932.496,E2 -8932.496} C_VEL
LIN {X 0,Y 442.991,Z 658.365,A -85,B 0,C 180,E1 -8933.367,E2 -8933.367} C_VEL
LIN {X 0,Y 442.567,Z 670.479,A -85,B 0,C 180,E1 -8934.262,E2 -8934.262} C_VEL
LIN {X 0,Y 442.035,Z 680.372,A -85,B 0,C 180,E1 -8935.174,E2 -8935.174} C_VEL
LIN {X 0,Y 441.576,Z 689.521,A -85,B 0,C 180,E1 -8936.21,E2 -8936.21} C_VEL
LIN {X 0,Y 441.045,Z 698.903,A -85,B 0,C 180,E1 -8937.524,E2 -8937.524} C_VEL
LIN {X 0,Y 440.547,Z 706.609,A -85,B 0,C 180,E1 -8938.853,E2 -8938.853} C_VEL
LIN {X 0,Y 440.205,Z 712.227,A -85,B 0,C 180,E1 -8940.042,E2 -8940.042} C_VEL
LIN {X 0,Y 439.889,Z 717.038,A -85,B 0,C 180,E1 -8941.282,E2 -8941.282} C_VEL
LIN {X 0,Y 439.625,Z 721.991,A -85,B 0,C 180,E1 -8942.925,E2 -8942.925} C_VEL
LIN {X 0,Y 439.44,Z 724.478,A -85,B 0,C 180,E1 -8944.039,E2 -8944.039} C_VEL
LIN {X 0,Y 439.281,Z 726.598,A -85,B 0,C 180,E1 -8945.32,E2 -8945.32} C_VEL
LIN {X 0,Y 439.199,Z 728.093,A -85,B 0,C 180,E1 -8946.861,E2 -8946.861} C_VEL
LIN {X 0,Y 439.256,Z 728.458,A -85,B 0,C 180,E1 -8948.608,E2 -8948.608} C_VEL
LIN {X 0,Y 439.29,Z 727.872,A -85,B 0,C 180,E1 -8949.832,E2 -8949.832} C_VEL
LIN {X 0,Y 439.391,Z 726.318,A -85,B 0,C 180,E1 -8951.257,E2 -8951.257} C_VEL
LIN {X 0,Y 439.608,Z 723.818,A -85,B 0,C 180,E1 -8952.659,E2 -8952.659} C_VEL
LIN {X 0,Y 439.867,Z 720.391,A -85,B 0,C 180,E1 -8954.029,E2 -8954.029} C_VEL
LIN {X 0,Y 440.199,Z 715.162,A -85,B 0,C 180,E1 -8955.595,E2 -8955.595} C_VEL
LIN {X 0,Y 440.706,Z 708.203,A -85,B 0,C 180,E1 -8957.187,E2 -8957.187} C_VEL
LIN {X 0,Y 441.207,Z 701.051,A -85,B 0,C 180,E1 -8958.475,E2 -8958.475} C_VEL
LIN {X 0,Y 441.742,Z 692.06,A -85,B 0,C 180,E1 -8959.789,E2 -8959.789} C_VEL
LIN {X 0,Y 442.388,Z 682.841,A -85,B 0,C 180,E1 -8960.874,E2 -8960.874} C_VEL
LIN {X 0,Y 442.829,Z 672.738,A -85,B 0,C 180,E1 -8961.843,E2 -8961.843} C_VEL
LIN {X 0,Y 443.264,Z 661.283,A -85,B 0,C 180,E1 -8962.715,E2 -8962.715} C_VEL
LIN {X 0,Y 443.115,Z 658.049,A -85,B 0,C 180,E1 -8962.937,E2 -8962.937} C_VEL
LIN {X 0,Y 439.41,Z 645.752,A -85,B 0,C 180,E1 -8963.797,E2 -8963.797} C_VEL
LIN {X 0,Y 439.373,Z 645.756,A -85,B 0,C 180,E1 -8967.054,E2 -8967.054} C_VEL
LIN {X 0,Y 439.383,Z 645.752,A -85,B 0,C 180,E1 -8970.274,E2 -8970.274} C_VEL
LIN {X 0,Y 439.429,Z 645.747,A -85,B 0,C 180,E1 -8973.396,E2 -8973.396} C_VEL
LIN {X 0,Y 439.384,Z 645.747,A -85,B 0,C 180,E1 -8976.43,E2 -8976.43} C_VEL
LIN {X 0,Y 439.389,Z 645.754,A -85,B 0,C 180,E1 -8979.397,E2 -8979.397} C_VEL
LIN {X 0,Y 439.433,Z 645.746,A -85,B 0,C 180,E1 -8982.31,E2 -8982.31} C_VEL
LIN {X 0,Y 439.453,Z 645.743,A -85,B 0,C 180,E1 -8985.174,E2 -8985.174} C_VEL
LIN {X 0,Y 439.485,Z 645.741,A -85,B 0,C 180,E1 -8988.001,E2 -8988.001} C_VEL
LIN {X 0,Y 439.549,Z 645.733,A -85,B 0,C 180,E1 -8991.726,E2 -8991.726} C_VEL
LIN {X 0,Y 439.622,Z 645.722,A -85,B 0,C 180,E1 -8994.496,E2 -8994.496} C_VEL
LIN {X 0,Y 439.637,Z 645.724,A -85,B 0,C 180,E1 -8998.168,E2 -8998.168} C_VEL
LIN {X 0,Y 439.765,Z 645.705,A -85,B 0,C 180,E1 -9000,E2 -9000} C_VEL
LIN {X 0,Y 439.658,Z 645.716,A -85,B 0,C 180,E1 -9002.749,E2 -9002.749} C_VEL
LIN {X 0,Y 439.619,Z 645.725,A -85,B 0,C 180,E1 -9006.425,E2 -9006.425} C_VEL
LIN {X 0,Y 439.502,Z 645.73,A -85,B 0,C 180,E1 -9009.202,E2 -9009.202} C_VEL
LIN {X 0,Y 439.467,Z 645.737,A -85,B 0,C 180,E1 -9012.938,E2 -9012.938} C_VEL
LIN {X 0,Y 439.449,Z 645.744,A -85,B 0,C 180,E1 -9016.349,E2 -9016.349} C_VEL
LIN {X 0,Y 439.404,Z 645.746,A -85,B 0,C 180,E1 -9019.626,E2 -9019.626} C_VEL
LIN {X 0,Y 439.367,Z 645.754,A -85,B 0,C 180,E1 -9022.576,E2 -9022.576} C_VEL
LIN {X 0,Y 439.407,Z 645.746,A -85,B 0,C 180,E1 -9025.585,E2 -9025.585} C_VEL
LIN {X 0,Y 439.419,Z 645.751,A -85,B 0,C 180,E1 -9028.674,E2 -9028.674} C_VEL
LIN {X 0,Y 439.372,Z 645.755,A -85,B 0,C 180,E1 -9032.03,E2 -9032.03} C_VEL
LIN {X 0,Y 439.396,Z 645.752,A -85,B 0,C 180,E1 -9035.34,E2 -9035.34} C_VEL
LIN {X 0,Y 439.381,Z 645.758,A -85,B 0,C 180,E1 -9038.595,E2 -9038.595} C_VEL
LIN {X 0,Y 439.391,Z 645.753,A -85,B 0,C 180,E1 -9041.257,E2 -9041.257} C_VEL
LIN {X 0,Y 439.404,Z 645.754,A -85,B 0,C 180,E1 -9044.729,E2 -9044.729} C_VEL
LIN {X 0,Y 439.423,Z 645.781,A -85,B 0,C 180,E1 -9048.235,E2 -9048.235} C_VEL
LIN {X 0,Y 441.305,Z 655.295,A -85,B 0,C 180,E1 -9051.293,E2 -9051.293} C_VEL
LIN {X 0,Y 442.349,Z 661.433,A -85,B 0,C 180,E1 -9053.146,E2 -9053.146} C_VEL
LIN {X 0,Y 441.923,Z 669.919,A -85,B 0,C 180,E1 -9055.492,E2 -9055.492} C_VEL
LIN {X 0,Y 441.224,Z 682.501,A -85,B 0,C 180,E1 -9058.823,E2 -9058.823} C_VEL
LIN {X 0,Y 440.604,Z 695.699,A -85,B 0,C 180,E1 -9062.188,E2 -9062.188} C_VEL
LIN {X 0,Y 440.083,Z 709.27,A -85,B 0,C 180,E1 -9065.544,E2 -9065.544} C_VEL
LIN {X 0,Y 439.609,Z 723.254,A -85,B 0,C 180,E1 -9068.918,E2 -9068.918} C_VEL
LIN {X 0,Y 439.293,Z 737.537,A -85,B 0,C 180,E1 -9072.303,E2 -9072.303} C_VEL
LIN {X 0,Y 439.175,Z 742.692,A -85,B 0,C 180,E1 -9073.515,E2 -9073.515} C_VEL
LIN {X 0,Y 440.604,Z 758.395,A -85,B 0,C 180,E1 -9073.992,E2 -9073.992} C_VEL
LIN {X 0,Y 442.049,Z 774.98,A -85,B 0,C 180,E1 -9074.673,E2 -9074.673} C_VEL
LIN {X 0,Y 441.596,Z 788.381,A -85,B 0,C 180,E1 -9075.365,E2 -9075.365} C_VEL
LIN {X 0,Y 440.969,Z 800.069,A -85,B 0,C 180,E1 -9076.168,E2 -9076.168} C_VEL
LIN {X 0,Y 440.39,Z 811.736,A -85,B 0,C 180,E1 -9077.207,E2 -9077.207} C_VEL
LIN {X 0,Y 439.902,Z 821.138,A -85,B 0,C 180,E1 -9078.246,E2 -9078.246} C_VEL
LIN {X 0,Y 439.394,Z 829.691,A -85,B 0,C 180,E1 -9079.4,E2 -9079.4} C_VEL
LIN {X 0,Y 438.998,Z 837.982,A -85,B 0,C 180,E1 -9080.787,E2 -9080.787} C_VEL
LIN {X 0,Y 438.717,Z 844.641,A -85,B 0,C 180,E1 -9082.174,E2 -9082.174} C_VEL
LIN {X 0,Y 438.51,Z 850.792,A -85,B 0,C 180,E1 -9083.825,E2 -9083.825} C_VEL
LIN {X 0,Y 438.434,Z 855.114,A -85,B 0,C 180,E1 -9085.402,E2 -9085.402} C_VEL
LIN {X 0,Y 438.383,Z 857.023,A -85,B 0,C 180,E1 -9086.323,E2 -9086.323} C_VEL
LIN {X 0,Y 438.424,Z 858.472,A -85,B 0,C 180,E1 -9087.243,E2 -9087.243} C_VEL
LIN {X 0,Y 438.375,Z 860.101,A -85,B 0,C 180,E1 -9089.081,E2 -9089.081} C_VEL
LIN {X 0,Y 438.38,Z 860.321,A -85,B 0,C 180,E1 -9090,E2 -9090} C_VEL
LIN {X 0,Y 438.372,Z 860.092,A -85,B 0,C 180,E1 -9090.918,E2 -9090.918} C_VEL
LIN {X 0,Y 438.423,Z 858.436,A -85,B 0,C 180,E1 -9092.756,E2 -9092.756} C_VEL
LIN {X 0,Y 438.376,Z 856.981,A -85,B 0,C 180,E1 -9093.676,E2 -9093.676} C_VEL
LIN {X 0,Y 438.482,Z 853.961,A -85,B 0,C 180,E1 -9095.057,E2 -9095.057} C_VEL
LIN {X 0,Y 438.506,Z 849.858,A -85,B 0,C 180,E1 -9096.441,E2 -9096.441} C_VEL
LIN {X 0,Y 438.74,Z 843.531,A -85,B 0,C 180,E1 -9098.057,E2 -9098.057} C_VEL
LIN {X 0,Y 439.054,Z 836.63,A -85,B 0,C 180,E1 -9099.443,E2 -9099.443} C_VEL
LIN {X 0,Y 439.44,Z 827.977,A -85,B 0,C 180,E1 -9100.831,E2 -9100.831} C_VEL
LIN {X 0,Y 439.986,Z 819.077,A -85,B 0,C 180,E1 -9101.984,E2 -9101.984} C_VEL
LIN {X 0,Y 440.486,Z 809.219,A -85,B 0,C 180,E1 -9103.031,E2 -9103.031} C_VEL
LIN {X 0,Y 441.035,Z 798.532,A -85,B 0,C 180,E1 -9103.946,E2 -9103.946} C_VEL
LIN {X 0,Y 441.622,Z 786.461,A -85,B 0,C 180,E1 -9104.751,E2 -9104.751} C_VEL
LIN {X 0,Y 442.109,Z 773.885,A -85,B 0,C 180,E1 -9105.383,E2 -9105.383} C_VEL
LIN {X 0,Y 440.524,Z 757.594,A -85,B 0,C 180,E1 -9106.058,E2 -9106.058} C_VEL
LIN {X 0,Y 439.167,Z 744.204,A -85,B 0,C 180,E1 -9106.464,E2 -9106.464} C_VEL
LIN {X 0,Y 439.539,Z 730.059,A -85,B 0,C 180,E1 -9109.863,E2 -9109.863} C_VEL
LIN {X 0,Y 440.051,Z 716.06,A -85,B 0,C 180,E1 -9113.283,E2 -9113.283} C_VEL
LIN {X 0,Y 440.606,Z 702.981,A -85,B 0,C 180,E1 -9116.526,E2 -9116.526} C_VEL
LIN {X 0,Y 441.202,Z 690.943,A -85,B 0,C 180,E1 -9119.59,E2 -9119.59} C_VEL
LIN {X 0,Y 441.854,Z 679.597,A -85,B 0,C 180,E1 -9122.541,E2 -9122.541} C_VEL
LIN {X 0,Y 442.539,Z 668.906,A -85,B 0,C 180,E1 -9125.403,E2 -9125.403} C_VEL
LIN {X 0,Y 442.746,Z 662.766,A -85,B 0,C 180,E1 -9127.098,E2 -9127.098} C_VEL
LIN {X 0,Y 440.84,Z 652.907,A -85,B 0,C 180,E1 -9130.072,E2 -9130.072} C_VEL
LIN {X 0,Y 439.404,Z 645.753,A -85,B 0,C 180,E1 -9132.36,E2 -9132.36} C_VEL
LIN {X 0,Y 439.406,Z 645.752,A -85,B 0,C 180,E1 -9135.271,E2 -9135.271} C_VEL
LIN {X 0,Y 439.402,Z 645.753,A -85,B 0,C 180,E1 -9138.74,E2 -9138.74} C_VEL
LIN {X 0,Y 439.39,Z 645.752,A -85,B 0,C 180,E1 -9141.604,E2 -9141.604} C_VEL
LIN {X 0,Y 439.397,Z 645.747,A -85,B 0,C 180,E1 -9144.844,E2 -9144.844} C_VEL
LIN {X 0,Y 439.37,Z 645.752,A -85,B 0,C 180,E1 -9148.139,E2 -9148.139} C_VEL
LIN {X 0,Y 439.421,Z 645.746,A -85,B 0,C 180,E1 -9151.327,E2 -9151.327} C_VEL
LIN {X 0,Y 439.401,Z 645.747,A -85,B 0,C 180,E1 -9154.415,E2 -9154.415} C_VEL
LIN {X 0,Y 439.361,Z 645.755,A -85,B 0,C 180,E1 -9157.424,E2 -9157.424} C_VEL
LIN {X 0,Y 439.436,Z 645.744,A -85,B 0,C 180,E1 -9160.662,E2 -9160.662} C_VEL
LIN {X 0,Y 439.457,Z 645.743,A -85,B 0,C 180,E1 -9164.224,E2 -9164.224} C_VEL
LIN {X 0,Y 439.507,Z 645.737,A -85,B 0,C 180,E1 -9168.002,E2 -9168.002} C_VEL
LIN {X 0,Y 439.543,Z 645.733,A -85,B 0,C 180,E1 -9171.726,E2 -9171.726} C_VEL
LIN {X 0,Y 439.616,Z 645.727,A -85,B 0,C 180,E1 -9174.496,E2 -9174.496} C_VEL
LIN {X 0,Y 439.63,Z 645.726,A -85,B 0,C 180,E1 -9178.168,E2 -9178.168} C_VEL
LIN {X 0,Y 439.758,Z 645.711,A -85,B 0,C 180,E1 -9180,E2 -9180} C_VEL
LIN {X 0,Y 439.65,Z 645.897,A -85,B 0,C 180,E1 -9182.061,E2 -9182.061} C_VEL
LIN {X 0,Y 441.063,Z 655.024,A -85,B 0,C 180,E1 -9184.57,E2 -9184.57} C_VEL
LIN {X 0,Y 441.167,Z 663.576,A -85,B 0,C 180,E1 -9186.862,E2 -9186.862} C_VEL
LIN {X 0,Y 440.959,Z 673.829,A -85,B 0,C 180,E1 -9189.634,E2 -9189.634} C_VEL
LIN {X 0,Y 440.761,Z 683.946,A -85,B 0,C 180,E1 -9192.431,E2 -9192.431} C_VEL
LIN {X 0,Y 440.448,Z 696.022,A -85,B 0,C 180,E1 -9195.739,E2 -9195.739} C_VEL
LIN {X 0,Y 440.16,Z 706.346,A -85,B 0,C 180,E1 -9198.623,E2 -9198.623} C_VEL
LIN {X 0,Y 439.8,Z 718.529,A -85,B 0,C 180,E1 -9202.055,E2 -9202.055} C_VEL
LIN {X 0,Y 439.549,Z 727.711,A -85,B 0,C 180,E1 -9204.627,E2 -9204.627} C_VEL
LIN {X 0,Y 442.05,Z 740.756,A -85,B 0,C 180,E1 -9205.075,E2 -9205.075} C_VEL
LIN {X 0,Y 442.814,Z 747.76,A -85,B 0,C 180,E1 -9205.374,E2 -9205.374} C_VEL
LIN {X 0,Y 442.364,Z 760.035,A -85,B 0,C 180,E1 -9205.97,E2 -9205.97} C_VEL
LIN {X 0,Y 441.745,Z 771.657,A -85,B 0,C 180,E1 -9206.717,E2 -9206.717} C_VEL
LIN {X 0,Y 441.134,Z 782.865,A -85,B 0,C 180,E1 -9207.646,E2 -9207.646} C_VEL
LIN {X 0,Y 440.524,Z 792.778,A -85,B 0,C 180,E1 -9208.665,E2 -9208.665} C_VEL
LIN {X 0,Y 439.924,Z 802.127,A -85,B 0,C 180,E1 -9209.847,E2 -9209.847} C_VEL
LIN {X 0,Y 439.462,Z 809.859,A -85,B 0,C 180,E1 -9211.048,E2 -9211.048} C_VEL
LIN {X 0,Y 439.057,Z 817.203,A -85,B 0,C 180,E1 -9212.448,E2 -9212.448} C_VEL
LIN {X 0,Y 438.801,Z 822.17,A -85,B 0,C 180,E1 -9213.609,E2 -9213.609} C_VEL
LIN {X 0,Y 438.513,Z 827.678,A -85,B 0,C 180,E1 -9215.238,E2 -9215.238} C_VEL
LIN {X 0,Y 438.34,Z 831.344,A -85,B 0,C 180,E1 -9216.712,E2 -9216.712} C_VEL
LIN {X 0,Y 438.223,Z 833.887,A -85,B 0,C 180,E1 -9218.203,E2 -9218.203} C_VEL
LIN {X 0,Y 438.114,Z 835.457,A -85,B 0,C 180,E1 -9219.916,E2 -9219.916} C_VEL
LIN {X 0,Y 438.095,Z 835.761,A -85,B 0,C 180,E1 -9221.127,E2 -9221.127} C_VEL
LIN {X 0,Y 438.086,Z 835.291,A -85,B 0,C 180,E1 -9222.444,E2 -9222.444} C_VEL
LIN {X 0,Y 438.171,Z 833.932,A -85,B 0,C 180,E1 -9223.8,E2 -9223.8} C_VEL
LIN {X 0,Y 438.312,Z 830.707,A -85,B 0,C 180,E1 -9225.616,E2 -9225.616} C_VEL
LIN {X 0,Y 438.502,Z 827.123,A -85,B 0,C 180,E1 -9226.991,E2 -9226.991} C_VEL
LIN {X 0,Y 438.744,Z 821.535,A -85,B 0,C 180,E1 -9228.602,E2 -9228.602} C_VEL
LIN {X 0,Y 439.071,Z 815.823,A -85,B 0,C 180,E1 -9229.891,E2 -9229.891} C_VEL
LIN {X 0,Y 439.473,Z 809.16,A -85,B 0,C 180,E1 -9231.122,E2 -9231.122} C_VEL
LIN {X 0,Y 439.943,Z 801.154,A -85,B 0,C 180,E1 -9232.337,E2 -9232.337} C_VEL
LIN {X 0,Y 440.535,Z 791.376,A -85,B 0,C 180,E1 -9233.541,E2 -9233.541} C_VEL
LIN {X 0,Y 441.181,Z 780.656,A -85,B 0,C 180,E1 -9234.609,E2 -9234.609} C_VEL
LIN {X 0,Y 441.738,Z 770.212,A -85,B 0,C 180,E1 -9235.441,E2 -9235.441} C_VEL
LIN {X 0,Y 442.399,Z 757.549,A -85,B 0,C 180,E1 -9236.22,E2 -9236.22} C_VEL
LIN {X 0,Y 442.664,Z 745.327,A -85,B 0,C 180,E1 -9236.789,E2 -9236.789} C_VEL
LIN {X 0,Y 440.535,Z 732.69,A -85,B 0,C 180,E1 -9237.272,E2 -9237.272} C_VEL
LIN {X 0,Y 439.481,Z 727.212,A -85,B 0,C 180,E1 -9237.453,E2 -9237.453} C_VEL
LIN {X 0,Y 439.973,Z 713.599,A -85,B 0,C 180,E1 -9241.367,E2 -9241.367} C_VEL
LIN {X 0,Y 440.276,Z 702.786,A -85,B 0,C 180,E1 -9244.47,E2 -9244.47} C_VEL
LIN {X 0,Y 440.661,Z 691.638,A -85,B 0,C 180,E1 -9247.673,E2 -9247.673} C_VEL
LIN {X 0,Y 440.998,Z 680.303,A -85,B 0,C 180,E1 -9250.932,E2 -9250.932} C_VEL
LIN {X 0,Y 441.274,Z 670.822,A -85,B 0,C 180,E1 -9253.66,E2 -9253.66} C_VEL
LIN {X 0,Y 440.738,Z 668.506,A -85,B 0,C 180,E1 -9254.361,E2 -9254.361} C_VEL
LIN {X 0,Y 438.114,Z 665.099,A -85,B 0,C 180,E1 -9255.523,E2 -9255.523} C_VEL
LIN {X 0,Y 434.933,Z 660.986,A -85,B 0,C 180,E1 -9256.939,E2 -9256.939} C_VEL
LIN {X 0,Y 434.514,Z 659.446,A -85,B 0,C 180,E1 -9257.42,E2 -9257.42} C_VEL
LIN {X 0,Y 433.729,Z 653.343,A -85,B 0,C 180,E1 -9259.261,E2 -9259.261} C_VEL
LIN {X 0,Y 432.504,Z 646.613,A -85,B 0,C 180,E1 -9261.356,E2 -9261.356} C_VEL
LIN {X 0,Y 432.599,Z 646.603,A -85,B 0,C 180,E1 -9264.407,E2 -9264.407} C_VEL
LIN {X 0,Y 432.607,Z 646.602,A -85,B 0,C 180,E1 -9268.139,E2 -9268.139} C_VEL
LIN {X 0,Y 432.735,Z 646.583,A -85,B 0,C 180,E1 -9270,E2 -9270} C_VEL
LIN {X 0,Y 432.607,Z 646.599,A -85,B 0,C 180,E1 -9272.794,E2 -9272.794} C_VEL
LIN {X 0,Y 432.57,Z 646.6,A -85,B 0,C 180,E1 -9276.531,E2 -9276.531} C_VEL
LIN {X 0,Y 432.446,Z 646.616,A -85,B 0,C 180,E1 -9279.353,E2 -9279.353} C_VEL
LIN {X 0,Y 432.447,Z 646.62,A -85,B 0,C 180,E1 -9282.812,E2 -9282.812} C_VEL
LIN {X 0,Y 432.414,Z 646.625,A -85,B 0,C 180,E1 -9286.479,E2 -9286.479} C_VEL
LIN {X 0,Y 432.34,Z 646.634,A -85,B 0,C 180,E1 -9289.961,E2 -9289.961} C_VEL
LIN {X 0,Y 432.352,Z 646.633,A -85,B 0,C 180,E1 -9292.234,E2 -9292.234} C_VEL
LIN {X 0,Y 436.068,Z 659.404,A -85,B 0,C 180,E1 -9293.147,E2 -9293.147} C_VEL
LIN {X 0,Y 435.74,Z 671.189,A -85,B 0,C 180,E1 -9294.033,E2 -9294.033} C_VEL
LIN {X 0,Y 435.169,Z 681.199,A -85,B 0,C 180,E1 -9294.966,E2 -9294.966} C_VEL
LIN {X 0,Y 434.636,Z 691.341,A -85,B 0,C 180,E1 -9296.144,E2 -9296.144} C_VEL
LIN {X 0,Y 434.082,Z 700.776,A -85,B 0,C 180,E1 -9297.509,E2 -9297.509} C_VEL
LIN {X 0,Y 433.556,Z 708.604,A -85,B 0,C 180,E1 -9298.914,E2 -9298.914} C_VEL
LIN {X 0,Y 433.195,Z 714.354,A -85,B 0,C 180,E1 -9300.194,E2 -9300.194} C_VEL
LIN {X 0,Y 432.807,Z 720.146,A -85,B 0,C 180,E1 -9301.837,E2 -9301.837} C_VEL
LIN {X 0,Y 432.529,Z 724.58,A -85,B 0,C 180,E1 -9303.536,E2 -9303.536} C_VEL
LIN {X 0,Y 432.341,Z 726.712,A -85,B 0,C 180,E1 -9304.677,E2 -9304.677} C_VEL
LIN {X 0,Y 432.245,Z 728.275,A -85,B 0,C 180,E1 -9305.827,E2 -9305.827} C_VEL
LIN {X 0,Y 432.177,Z 729.295,A -85,B 0,C 180,E1 -9307.172,E2 -9307.172} C_VEL
LIN {X 0,Y 432.234,Z 729.48,A -85,B 0,C 180,E1 -9308.697,E2 -9308.697} C_VEL
LIN {X 0,Y 432.334,Z 728.283,A -85,B 0,C 180,E1 -9310.56,E2 -9310.56} C_VEL
LIN {X 0,Y 432.56,Z 725.568,A -85,B 0,C 180,E1 -9312.398,E2 -9312.398} C_VEL
LIN {X 0,Y 432.917,Z 721.036,A -85,B 0,C 180,E1 -9314.272,E2 -9314.272} C_VEL
LIN {X 0,Y 433.274,Z 716.03,A -85,B 0,C 180,E1 -9315.774,E2 -9315.774} C_VEL
LIN {X 0,Y 433.757,Z 710.319,A -85,B 0,C 180,E1 -9317.117,E2 -9317.117} C_VEL
LIN {X 0,Y 434.221,Z 703.466,A -85,B 0,C 180,E1 -9318.425,E2 -9318.425} C_VEL
LIN {X 0,Y 434.802,Z 695.07,A -85,B 0,C 180,E1 -9319.718,E2 -9319.718} C_VEL
LIN {X 0,Y 435.491,Z 684.729,A -85,B 0,C 180,E1 -9320.995,E2 -9320.995} C_VEL
LIN {X 0,Y 436.024,Z 674.135,A -85,B 0,C 180,E1 -9322.044,E2 -9322.044} C_VEL
LIN {X 0,Y 436.497,Z 662.727,A -85,B 0,C 180,E1 -9322.931,E2 -9322.931} C_VEL
LIN {X 0,Y 436.4,Z 659.813,A -85,B 0,C 180,E1 -9323.138,E2 -9323.138} C_VEL
LIN {X 0,Y 432.893,Z 648.573,A -85,B 0,C 180,E1 -9323.948,E2 -9323.948} C_VEL
LIN {X 0,Y 432.358,Z 646.63,A -85,B 0,C 180,E1 -9324.077,E2 -9324.077} C_VEL
LIN {X 0,Y 432.34,Z 646.63,A -85,B 0,C 180,E1 -9326.448,E2 -9326.448} C_VEL
LIN {X 0,Y 432.346,Z 646.634,A -85,B 0,C 180,E1 -9329.74,E2 -9329.74} C_VEL
LIN {X 0,Y 432.391,Z 646.623,A -85,B 0,C 180,E1 -9332.928,E2 -9332.928} C_VEL
LIN {X 0,Y 432.368,Z 646.624,A -85,B 0,C 180,E1 -9336.023,E2 -9336.023} C_VEL
LIN {X 0,Y 432.351,Z 646.629,A -85,B 0,C 180,E1 -9339.046,E2 -9339.046} C_VEL
LIN {X 0,Y 432.38,Z 646.628,A -85,B 0,C 180,E1 -9342.011,E2 -9342.011} C_VEL
LIN {X 0,Y 432.403,Z 646.621,A -85,B 0,C 180,E1 -9344.927,E2 -9344.927} C_VEL
LIN {X 0,Y 432.46,Z 646.619,A -85,B 0,C 180,E1 -9347.804,E2 -9347.804} C_VEL
LIN {X 0,Y 432.493,Z 646.611,A -85,B 0,C 180,E1 -9351.59,E2 -9351.59} C_VEL
LIN {X 0,Y 432.599,Z 646.598,A -85,B 0,C 180,E1 -9354.406,E2 -9354.406} C_VEL
LIN {X 0,Y 432.607,Z 646.599,A -85,B 0,C 180,E1 -9358.138,E2 -9358.138} C_VEL
LIN {X 0,Y 432.735,Z 646.58,A -85,B 0,C 180,E1 -9360,E2 -9360} C_VEL
LIN {X 0,Y 432.607,Z 646.594,A -85,B 0,C 180,E1 -9362.794,E2 -9362.794} C_VEL
LIN {X 0,Y 432.574,Z 646.601,A -85,B 0,C 180,E1 -9366.53,E2 -9366.53} C_VEL
LIN {X 0,Y 432.445,Z 646.609,A -85,B 0,C 180,E1 -9369.353,E2 -9369.353} C_VEL
LIN {X 0,Y 432.432,Z 646.614,A -85,B 0,C 180,E1 -9372.804,E2 -9372.804} C_VEL
LIN {X 0,Y 432.414,Z 646.619,A -85,B 0,C 180,E1 -9376.479,E2 -9376.479} C_VEL
LIN {X 0,Y 432.341,Z 646.628,A -85,B 0,C 180,E1 -9379.961,E2 -9379.961} C_VEL
LIN {X 0,Y 432.321,Z 646.63,A -85,B 0,C 180,E1 -9382.964,E2 -9382.964} C_VEL
LIN {X 0,Y 432.366,Z 646.626,A -85,B 0,C 180,E1 -9386.033,E2 -9386.033} C_VEL
LIN {X 0,Y 432.345,Z 646.629,A -85,B 0,C 180,E1 -9389.188,E2 -9389.188} C_VEL
LIN {X 0,Y 432.325,Z 646.635,A -85,B 0,C 180,E1 -9392.443,E2 -9392.443} C_VEL
LIN {X 0,Y 432.346,Z 646.63,A -85,B 0,C 180,E1 -9395.632,E2 -9395.632} C_VEL
LIN {X 0,Y 432.349,Z 646.63,A -85,B 0,C 180,E1 -9399.343,E2 -9399.343} C_VEL
LIN {X 0,Y 432.336,Z 646.631,A -85,B 0,C 180,E1 -9401.797,E2 -9401.797} C_VEL
LIN {X 0,Y 432.336,Z 646.633,A -85,B 0,C 180,E1 -9404.347,E2 -9404.347} C_VEL
LIN {X 0,Y 432.373,Z 646.689,A -85,B 0,C 180,E1 -9407.894,E2 -9407.894} C_VEL
LIN {X 0,Y 434.148,Z 655.609,A -85,B 0,C 180,E1 -9410.851,E2 -9410.851} C_VEL
LIN {X 0,Y 435.312,Z 662.019,A -85,B 0,C 180,E1 -9412.841,E2 -9412.841} C_VEL
LIN {X 0,Y 435.286,Z 666.498,A -85,B 0,C 180,E1 -9414.134,E2 -9414.134} C_VEL
LIN {X 0,Y 434.545,Z 677.82,A -85,B 0,C 180,E1 -9417.247,E2 -9417.247} C_VEL
LIN {X 0,Y 433.834,Z 690.73,A -85,B 0,C 180,E1 -9420.656,E2 -9420.656} C_VEL
LIN {X 0,Y 433.259,Z 703.96,A -85,B 0,C 180,E1 -9424.025,E2 -9424.025} C_VEL
LIN {X 0,Y 432.795,Z 716.162,A -85,B 0,C 180,E1 -9427.062,E2 -9427.062} C_VEL
LIN {X 0,Y 432.346,Z 731.391,A -85,B 0,C 180,E1 -9430.783,E2 -9430.783} C_VEL
LIN {X 0,Y 432.093,Z 741.585,A -85,B 0,C 180,E1 -9433.231,E2 -9433.231} C_VEL
LIN {X 0,Y 433.485,Z 756.253,A -85,B 0,C 180,E1 -9433.68,E2 -9433.68} C_VEL
LIN {X 0,Y 434.988,Z 772.553,A -85,B 0,C 180,E1 -9434.328,E2 -9434.328} C_VEL
LIN {X 0,Y 435.071,Z 778.502,A -85,B 0,C 180,E1 -9434.601,E2 -9434.601} C_VEL
LIN {X 0,Y 434.607,Z 789.992,A -85,B 0,C 180,E1 -9435.244,E2 -9435.244} C_VEL
LIN {X 0,Y 433.997,Z 800.928,A -85,B 0,C 180,E1 -9436.036,E2 -9436.036} C_VEL
LIN {X 0,Y 433.423,Z 811.482,A -85,B 0,C 180,E1 -9436.998,E2 -9436.998} C_VEL
LIN {X 0,Y 432.915,Z 820.892,A -85,B 0,C 180,E1 -9438.054,E2 -9438.054} C_VEL
LIN {X 0,Y 432.382,Z 829.457,A -85,B 0,C 180,E1 -9439.226,E2 -9439.226} C_VEL
LIN {X 0,Y 431.953,Z 837.755,A -85,B 0,C 180,E1 -9440.636,E2 -9440.636} C_VEL
LIN {X 0,Y 431.638,Z 844.42,A -85,B 0,C 180,E1 -9442.044,E2 -9442.044} C_VEL
LIN {X 0,Y 431.463,Z 849.959,A -85,B 0,C 180,E1 -9443.524,E2 -9443.524} C_VEL
LIN {X 0,Y 431.407,Z 853.808,A -85,B 0,C 180,E1 -9444.859,E2 -9444.859} C_VEL
LIN {X 0,Y 431.285,Z 856.817,A -85,B 0,C 180,E1 -9446.262,E2 -9446.262} C_VEL
